   DATA[1858,0] := 2.531467;
   DATA[1858,1] := 861.0878;
   DATA[1858,2] := 2.0;
   DATA[1858,3] := 2.0;
   DATA[1858,4] := 263.362;
   DATA[1858,5] := 8.398359;
   DATA[1858,6] := 333.3761;
   DATA[1858,7] := 2.469228;
   DATA[1858,8] := 2.0;
   DATA[1858,9] := 2.0;
   DATA[1858,10] := 2.0;
   DATA[1858,11] := 19.80601;
   DATA[1858,12] := 2.208756;
   DATA[1858,13] := 790.5024;
   DATA[1858,14] := 1.0;
   DATA[1858,15] := 2.0;
   DATA[1858,16] := 1.0;
   DATA[1858,17] := 1.0;
   DATA[1858,18] := 1.0;
   DATA[1858,19] := 2.0;
   DATA[1858,20] := 148.808;
   DATA[1858,21] := 154.4476;
   DATA[1858,22] := 1.711723;
   DATA[1858,23] := 818.2517;
   DATA[1858,24] := 2.0;
   DATA[1858,25] := 2.0;
   DATA[1858,26] := 7.874135;
   DATA[1858,27] := 143.5529;
   DATA[1858,28] := 262.3686;
   DATA[1858,29] := 12.15073;
   DATA[1858,30] := 1.72161;
   DATA[1858,31] := 1.282567;
   DATA[1858,32] := 0.7355248;
   DATA[1858,33] := 0.3084265;
   DATA[1858,34] := 2.0;
   DATA[1858,35] := 249.8238;
   DATA[1858,36] := 1.69801;
   DATA[1858,37] := 188.6856;
   DATA[1858,38] := 0.000128152;
   DATA[1858,39] := 1.0;
   DATA[1858,40] := 1.0;
   DATA[1859,0] := 2.567658;
   DATA[1859,1] := 861.0093;
   DATA[1859,2] := 2.0;
   DATA[1859,3] := 2.0;
   DATA[1859,4] := 263.362;
   DATA[1859,5] := 8.398039;
   DATA[1859,6] := 333.4786;
   DATA[1859,7] := 2.469228;
   DATA[1859,8] := 2.0;
   DATA[1859,9] := 2.0;
   DATA[1859,10] := 2.0;
   DATA[1859,11] := 19.80601;
   DATA[1859,12] := 2.208756;
   DATA[1859,13] := 790.7027;
   DATA[1859,14] := 1.0;
   DATA[1859,15] := 2.0;
   DATA[1859,16] := 1.0;
   DATA[1859,17] := 1.0;
   DATA[1859,18] := 1.0;
   DATA[1859,19] := 2.0;
   DATA[1859,20] := 148.808;
   DATA[1859,21] := 154.4476;
   DATA[1859,22] := 1.710313;
   DATA[1859,23] := 818.2902;
   DATA[1859,24] := 2.0;
   DATA[1859,25] := 2.0;
   DATA[1859,26] := 7.874135;
   DATA[1859,27] := 143.5529;
   DATA[1859,28] := 262.3686;
   DATA[1859,29] := 12.15073;
   DATA[1859,30] := 1.72161;
   DATA[1859,31] := 1.273473;
   DATA[1859,32] := 0.7355248;
   DATA[1859,33] := 0.3084265;
   DATA[1859,34] := 2.0;
   DATA[1859,35] := 249.8238;
   DATA[1859,36] := 1.69801;
   DATA[1859,37] := 188.6856;
   DATA[1859,38] := 0.000128152;
   DATA[1859,39] := 1.0;
   DATA[1859,40] := 1.0;
   DATA[1860,0] := 2.606091;
   DATA[1860,1] := 860.6167;
   DATA[1860,2] := 2.0;
   DATA[1860,3] := 2.0;
   DATA[1860,4] := 263.2979;
   DATA[1860,5] := 8.393873;
   DATA[1860,6] := 333.4786;
   DATA[1860,7] := 2.469228;
   DATA[1860,8] := 2.0;
   DATA[1860,9] := 2.0;
   DATA[1860,10] := 2.0;
   DATA[1860,11] := 19.80601;
   DATA[1860,12] := 2.210294;
   DATA[1860,13] := 790.7027;
   DATA[1860,14] := 1.0;
   DATA[1860,15] := 2.0;
   DATA[1860,16] := 1.0;
   DATA[1860,17] := 1.0;
   DATA[1860,18] := 1.0;
   DATA[1860,19] := 2.0;
   DATA[1860,20] := 148.808;
   DATA[1860,21] := 154.4476;
   DATA[1860,22] := 1.710313;
   DATA[1860,23] := 818.2517;
   DATA[1860,24] := 2.0;
   DATA[1860,25] := 2.0;
   DATA[1860,26] := 7.874135;
   DATA[1860,27] := 143.5529;
   DATA[1860,28] := 262.3686;
   DATA[1860,29] := 12.15073;
   DATA[1860,30] := 1.723532;
   DATA[1860,31] := 1.277187;
   DATA[1860,32] := 0.7355248;
   DATA[1860,33] := 0.3084265;
   DATA[1860,34] := 2.0;
   DATA[1860,35] := 250.0961;
   DATA[1860,36] := 1.69801;
   DATA[1860,37] := 189.006;
   DATA[1860,38] := 0.000128152;
   DATA[1860,39] := 1.0;
   DATA[1860,40] := 1.0;
   DATA[1861,0] := 2.633635;
   DATA[1861,1] := 860.8522;
   DATA[1861,2] := 2.0;
   DATA[1861,3] := 2.0;
   DATA[1861,4] := 263.0095;
   DATA[1861,5] := 8.393873;
   DATA[1861,6] := 333.4786;
   DATA[1861,7] := 2.469228;
   DATA[1861,8] := 2.0;
   DATA[1861,9] := 2.0;
   DATA[1861,10] := 2.0;
   DATA[1861,11] := 19.73238;
   DATA[1861,12] := 2.210294;
   DATA[1861,13] := 790.7828;
   DATA[1861,14] := 1.0;
   DATA[1861,15] := 2.0;
   DATA[1861,16] := 1.0;
   DATA[1861,17] := 1.0;
   DATA[1861,18] := 1.0;
   DATA[1861,19] := 2.0;
   DATA[1861,20] := 148.808;
   DATA[1861,21] := 154.5245;
   DATA[1861,22] := 1.710313;
   DATA[1861,23] := 817.9441;
   DATA[1861,24] := 2.0;
   DATA[1861,25] := 2.0;
   DATA[1861,26] := 7.874135;
   DATA[1861,27] := 143.5529;
   DATA[1861,28] := 262.3686;
   DATA[1861,29] := 12.15073;
   DATA[1861,30] := 1.724045;
   DATA[1861,31] := 1.275522;
   DATA[1861,32] := 0.7355248;
   DATA[1861,33] := 0.3084265;
   DATA[1861,34] := 2.0;
   DATA[1861,35] := 250.0961;
   DATA[1861,36] := 1.69801;
   DATA[1861,37] := 189.006;
   DATA[1861,38] := 0.000128152;
   DATA[1861,39] := 1.0;
   DATA[1861,40] := 1.0;
   DATA[1862,0] := 2.654133;
   DATA[1862,1] := 860.8915;
   DATA[1862,2] := 2.0;
   DATA[1862,3] := 2.0;
   DATA[1862,4] := 262.9454;
   DATA[1862,5] := 8.393873;
   DATA[1862,6] := 333.4786;
   DATA[1862,7] := 2.469228;
   DATA[1862,8] := 2.0;
   DATA[1862,9] := 2.0;
   DATA[1862,10] := 2.0;
   DATA[1862,11] := 19.73238;
   DATA[1862,12] := 2.207731;
   DATA[1862,13] := 791.4637;
   DATA[1862,14] := 1.0;
   DATA[1862,15] := 2.0;
   DATA[1862,16] := 1.0;
   DATA[1862,17] := 1.0;
   DATA[1862,18] := 1.0;
   DATA[1862,19] := 2.0;
   DATA[1862,20] := 148.808;
   DATA[1862,21] := 154.5245;
   DATA[1862,22] := 1.710313;
   DATA[1862,23] := 818.4055;
   DATA[1862,24] := 2.0;
   DATA[1862,25] := 2.0;
   DATA[1862,26] := 7.874135;
   DATA[1862,27] := 143.5529;
   DATA[1862,28] := 262.3686;
   DATA[1862,29] := 12.15073;
   DATA[1862,30] := 1.724045;
   DATA[1862,31] := 1.278596;
   DATA[1862,32] := 0.7355248;
   DATA[1862,33] := 0.3084265;
   DATA[1862,34] := 2.0;
   DATA[1862,35] := 250.0961;
   DATA[1862,36] := 1.69801;
   DATA[1862,37] := 189.006;
   DATA[1862,38] := 0.000128152;
   DATA[1862,39] := 1.0;
   DATA[1862,40] := 1.0;
   DATA[1863,0] := 2.664382;
   DATA[1863,1] := 860.8915;
   DATA[1863,2] := 2.0;
   DATA[1863,3] := 2.0;
   DATA[1863,4] := 262.9454;
   DATA[1863,5] := 8.393873;
   DATA[1863,6] := 333.4786;
   DATA[1863,7] := 2.469228;
   DATA[1863,8] := 2.0;
   DATA[1863,9] := 2.0;
   DATA[1863,10] := 2.0;
   DATA[1863,11] := 19.73238;
   DATA[1863,12] := 2.20581;
   DATA[1863,13] := 791.664;
   DATA[1863,14] := 1.0;
   DATA[1863,15] := 2.0;
   DATA[1863,16] := 1.0;
   DATA[1863,17] := 1.0;
   DATA[1863,18] := 1.0;
   DATA[1863,19] := 2.0;
   DATA[1863,20] := 148.808;
   DATA[1863,21] := 154.5245;
   DATA[1863,22] := 1.710313;
   DATA[1863,23] := 818.444;
   DATA[1863,24] := 2.0;
   DATA[1863,25] := 2.0;
   DATA[1863,26] := 7.874135;
   DATA[1863,27] := 143.5529;
   DATA[1863,28] := 262.3686;
   DATA[1863,29] := 12.15073;
   DATA[1863,30] := 1.724045;
   DATA[1863,31] := 1.291405;
   DATA[1863,32] := 0.7355248;
   DATA[1863,33] := 0.3084265;
   DATA[1863,34] := 2.0;
   DATA[1863,35] := 250.0961;
   DATA[1863,36] := 1.69801;
   DATA[1863,37] := 189.006;
   DATA[1863,38] := 0.000128152;
   DATA[1863,39] := 1.0;
   DATA[1863,40] := 1.0;
   DATA[1864,0] := 2.664382;
   DATA[1864,1] := 861.127;
   DATA[1864,2] := 2.0;
   DATA[1864,3] := 2.0;
   DATA[1864,4] := 262.9454;
   DATA[1864,5] := 8.393873;
   DATA[1864,6] := 333.4786;
   DATA[1864,7] := 2.467818;
   DATA[1864,8] := 2.0;
   DATA[1864,9] := 2.0;
   DATA[1864,10] := 2.0;
   DATA[1864,11] := 19.73238;
   DATA[1864,12] := 2.20581;
   DATA[1864,13] := 791.9044;
   DATA[1864,14] := 1.0;
   DATA[1864,15] := 2.0;
   DATA[1864,16] := 1.0;
   DATA[1864,17] := 1.0;
   DATA[1864,18] := 1.0;
   DATA[1864,19] := 2.0;
   DATA[1864,20] := 148.808;
   DATA[1864,21] := 154.5245;
   DATA[1864,22] := 1.710313;
   DATA[1864,23] := 818.6747;
   DATA[1864,24] := 2.0;
   DATA[1864,25] := 2.0;
   DATA[1864,26] := 7.874135;
   DATA[1864,27] := 143.5529;
   DATA[1864,28] := 262.3045;
   DATA[1864,29] := 12.15073;
   DATA[1864,30] := 1.724045;
   DATA[1864,31] := 1.28641;
   DATA[1864,32] := 0.7355248;
   DATA[1864,33] := 0.3084265;
   DATA[1864,34] := 2.0;
   DATA[1864,35] := 250.0961;
   DATA[1864,36] := 1.537821;
   DATA[1864,37] := 188.8618;
   DATA[1864,38] := 0.000128152;
   DATA[1864,39] := 1.0;
   DATA[1864,40] := 1.0;
   DATA[1865,0] := 2.63876;
   DATA[1865,1] := 861.2055;
   DATA[1865,2] := 2.0;
   DATA[1865,3] := 2.0;
   DATA[1865,4] := 262.9454;
   DATA[1865,5] := 8.393873;
   DATA[1865,6] := 333.6837;
   DATA[1865,7] := 2.467818;
   DATA[1865,8] := 2.0;
   DATA[1865,9] := 2.0;
   DATA[1865,10] := 2.0;
   DATA[1865,11] := 19.73238;
   DATA[1865,12] := 2.208244;
   DATA[1865,13] := 791.9044;
   DATA[1865,14] := 1.0;
   DATA[1865,15] := 2.0;
   DATA[1865,16] := 1.0;
   DATA[1865,17] := 1.0;
   DATA[1865,18] := 1.0;
   DATA[1865,19] := 2.0;
   DATA[1865,20] := 148.808;
   DATA[1865,21] := 154.5245;
   DATA[1865,22] := 1.710698;
   DATA[1865,23] := 819.213;
   DATA[1865,24] := 2.0;
   DATA[1865,25] := 2.0;
   DATA[1865,26] := 7.874135;
   DATA[1865,27] := 143.5529;
   DATA[1865,28] := 262.1764;
   DATA[1865,29] := 12.15073;
   DATA[1865,30] := 1.724045;
   DATA[1865,31] := 1.289356;
   DATA[1865,32] := 0.7355248;
   DATA[1865,33] := 0.3084265;
   DATA[1865,34] := 2.0;
   DATA[1865,35] := 250.0961;
   DATA[1865,36] := 1.537821;
   DATA[1865,37] := 188.6856;
   DATA[1865,38] := 0.000128152;
   DATA[1865,39] := 1.0;
   DATA[1865,40] := 1.0;
   DATA[1866,0] := 2.630753;
   DATA[1866,1] := 860.8915;
   DATA[1866,2] := 2.0;
   DATA[1866,3] := 2.0;
   DATA[1866,4] := 262.9454;
   DATA[1866,5] := 8.393873;
   DATA[1866,6] := 333.6837;
   DATA[1866,7] := 2.467818;
   DATA[1866,8] := 2.0;
   DATA[1866,9] := 2.0;
   DATA[1866,10] := 2.0;
   DATA[1866,11] := 19.73238;
   DATA[1866,12] := 2.209397;
   DATA[1866,13] := 792.0646;
   DATA[1866,14] := 1.0;
   DATA[1866,15] := 2.0;
   DATA[1866,16] := 1.0;
   DATA[1866,17] := 1.0;
   DATA[1866,18] := 1.0;
   DATA[1866,19] := 2.0;
   DATA[1866,20] := 148.808;
   DATA[1866,21] := 154.6526;
   DATA[1866,22] := 1.712107;
   DATA[1866,23] := 818.9823;
   DATA[1866,24] := 2.0;
   DATA[1866,25] := 2.0;
   DATA[1866,26] := 7.874135;
   DATA[1866,27] := 143.5529;
   DATA[1866,28] := 262.1764;
   DATA[1866,29] := 12.15073;
   DATA[1866,30] := 1.724045;
   DATA[1866,31] := 1.291789;
   DATA[1866,32] := 0.7355248;
   DATA[1866,33] := 0.3084265;
   DATA[1866,34] := 2.0;
   DATA[1866,35] := 250.0961;
   DATA[1866,36] := 1.762086;
   DATA[1866,37] := 188.6856;
   DATA[1866,38] := 0.000128152;
   DATA[1866,39] := 1.0;
   DATA[1866,40] := 1.0;
   DATA[1867,0] := 2.625628;
   DATA[1867,1] := 861.0878;
   DATA[1867,2] := 2.0;
   DATA[1867,3] := 2.0;
   DATA[1867,4] := 262.9454;
   DATA[1867,5] := 8.393873;
   DATA[1867,6] := 333.6837;
   DATA[1867,7] := 2.467818;
   DATA[1867,8] := 2.0;
   DATA[1867,9] := 2.0;
   DATA[1867,10] := 2.0;
   DATA[1867,11] := 19.69396;
   DATA[1867,12] := 2.209397;
   DATA[1867,13] := 792.3449;
   DATA[1867,14] := 1.0;
   DATA[1867,15] := 2.0;
   DATA[1867,16] := 1.0;
   DATA[1867,17] := 1.0;
   DATA[1867,18] := 1.0;
   DATA[1867,19] := 2.0;
   DATA[1867,20] := 148.808;
   DATA[1867,21] := 154.6526;
   DATA[1867,22] := 1.714286;
   DATA[1867,23] := 819.1746;
   DATA[1867,24] := 2.0;
   DATA[1867,25] := 2.0;
   DATA[1867,26] := 7.874135;
   DATA[1867,27] := 143.5529;
   DATA[1867,28] := 262.1764;
   DATA[1867,29] := 12.15073;
   DATA[1867,30] := 1.723789;
   DATA[1867,31] := 1.293455;
   DATA[1867,32] := 0.7355248;
   DATA[1867,33] := 0.3084265;
   DATA[1867,34] := 2.0;
   DATA[1867,35] := 250.0961;
   DATA[1867,36] := 1.762086;
   DATA[1867,37] := 188.6856;
   DATA[1867,38] := 0.000128152;
   DATA[1867,39] := 1.0;
   DATA[1867,40] := 1.0;
   DATA[1868,0] := 2.617942;
   DATA[1868,1] := 860.813;
   DATA[1868,2] := 2.0;
   DATA[1868,3] := 2.0;
   DATA[1868,4] := 262.9454;
   DATA[1868,5] := 8.393873;
   DATA[1868,6] := 333.6837;
   DATA[1868,7] := 2.467818;
   DATA[1868,8] := 2.0;
   DATA[1868,9] := 2.0;
   DATA[1868,10] := 2.0;
   DATA[1868,11] := 19.69396;
   DATA[1868,12] := 2.209397;
   DATA[1868,13] := 792.3049;
   DATA[1868,14] := 1.0;
   DATA[1868,15] := 2.0;
   DATA[1868,16] := 1.0;
   DATA[1868,17] := 1.0;
   DATA[1868,18] := 1.0;
   DATA[1868,19] := 2.0;
   DATA[1868,20] := 148.808;
   DATA[1868,21] := 154.6526;
   DATA[1868,22] := 1.714926;
   DATA[1868,23] := 819.0977;
   DATA[1868,24] := 2.0;
   DATA[1868,25] := 2.0;
   DATA[1868,26] := 7.874135;
   DATA[1868,27] := 143.5529;
   DATA[1868,28] := 262.1764;
   DATA[1868,29] := 12.15073;
   DATA[1868,30] := 1.721866;
   DATA[1868,31] := 1.302165;
   DATA[1868,32] := 0.7355248;
   DATA[1868,33] := 0.3084265;
   DATA[1868,34] := 2.0;
   DATA[1868,35] := 249.9359;
   DATA[1868,36] := 1.762086;
   DATA[1868,37] := 188.8618;
   DATA[1868,38] := 0.000128152;
   DATA[1868,39] := 1.0;
   DATA[1868,40] := 1.0;
   DATA[1869,0] := 2.596483;
   DATA[1869,1] := 860.6167;
   DATA[1869,2] := 2.0;
   DATA[1869,3] := 2.0;
   DATA[1869,4] := 262.9454;
   DATA[1869,5] := 8.393873;
   DATA[1869,6] := 333.6837;
   DATA[1869,7] := 2.467818;
   DATA[1869,8] := 2.0;
   DATA[1869,9] := 2.0;
   DATA[1869,10] := 2.0;
   DATA[1869,11] := 19.71637;
   DATA[1869,12] := 2.209397;
   DATA[1869,13] := 792.6653;
   DATA[1869,14] := 1.0;
   DATA[1869,15] := 2.0;
   DATA[1869,16] := 1.0;
   DATA[1869,17] := 1.0;
   DATA[1869,18] := 1.0;
   DATA[1869,19] := 2.0;
   DATA[1869,20] := 148.808;
   DATA[1869,21] := 154.6526;
   DATA[1869,22] := 1.714926;
   DATA[1869,23] := 819.6744;
   DATA[1869,24] := 2.0;
   DATA[1869,25] := 2.0;
   DATA[1869,26] := 7.874135;
   DATA[1869,27] := 143.5529;
   DATA[1869,28] := 262.3366;
   DATA[1869,29] := 12.15073;
   DATA[1869,30] := 1.721866;
   DATA[1869,31] := 1.29512;
   DATA[1869,32] := 0.7355248;
   DATA[1869,33] := 0.3084265;
   DATA[1869,34] := 2.0;
   DATA[1869,35] := 249.9359;
   DATA[1869,36] := 1.762086;
   DATA[1869,37] := 188.8618;
   DATA[1869,38] := 0.000128152;
   DATA[1869,39] := 1.0;
   DATA[1869,40] := 1.0;
   DATA[1870,0] := 2.58111;
   DATA[1870,1] := 860.4205;
   DATA[1870,2] := 2.0;
   DATA[1870,3] := 2.0;
   DATA[1870,4] := 262.9454;
   DATA[1870,5] := 8.392271;
   DATA[1870,6] := 333.4786;
   DATA[1870,7] := 2.46769;
   DATA[1870,8] := 2.0;
   DATA[1870,9] := 2.0;
   DATA[1870,10] := 2.0;
   DATA[1870,11] := 19.73878;
   DATA[1870,12] := 2.209397;
   DATA[1870,13] := 793.146;
   DATA[1870,14] := 1.0;
   DATA[1870,15] := 2.0;
   DATA[1870,16] := 1.0;
   DATA[1870,17] := 1.0;
   DATA[1870,18] := 1.0;
   DATA[1870,19] := 2.0;
   DATA[1870,20] := 148.808;
   DATA[1870,21] := 154.6526;
   DATA[1870,22] := 1.714926;
   DATA[1870,23] := 819.5591;
   DATA[1870,24] := 2.0;
   DATA[1870,25] := 2.0;
   DATA[1870,26] := 7.874135;
   DATA[1870,27] := 143.5529;
   DATA[1870,28] := 262.3366;
   DATA[1870,29] := 12.15073;
   DATA[1870,30] := 1.724045;
   DATA[1870,31] := 1.292174;
   DATA[1870,32] := 0.7355248;
   DATA[1870,33] := 0.3084265;
   DATA[1870,34] := 2.0;
   DATA[1870,35] := 249.9359;
   DATA[1870,36] := 1.762086;
   DATA[1870,37] := 188.8618;
   DATA[1870,38] := 0.000128152;
   DATA[1870,39] := 1.0;
   DATA[1870,40] := 1.0;
   DATA[1871,0] := 2.55837;
   DATA[1871,1] := 860.2634;
   DATA[1871,2] := 2.0;
   DATA[1871,3] := 2.0;
   DATA[1871,4] := 262.9454;
   DATA[1871,5] := 8.39163;
   DATA[1871,6] := 333.4273;
   DATA[1871,7] := 2.466024;
   DATA[1871,8] := 2.0;
   DATA[1871,9] := 2.0;
   DATA[1871,10] := 2.0;
   DATA[1871,11] := 19.73878;
   DATA[1871,12] := 2.21119;
   DATA[1871,13] := 793.0659;
   DATA[1871,14] := 1.0;
   DATA[1871,15] := 2.0;
   DATA[1871,16] := 1.0;
   DATA[1871,17] := 1.0;
   DATA[1871,18] := 1.0;
   DATA[1871,19] := 2.0;
   DATA[1871,20] := 148.808;
   DATA[1871,21] := 154.6526;
   DATA[1871,22] := 1.717105;
   DATA[1871,23] := 819.213;
   DATA[1871,24] := 2.0;
   DATA[1871,25] := 2.0;
   DATA[1871,26] := 7.874135;
   DATA[1871,27] := 143.5529;
   DATA[1871,28] := 262.3366;
   DATA[1871,29] := 12.15073;
   DATA[1871,30] := 1.724173;
   DATA[1871,31] := 1.290637;
   DATA[1871,32] := 0.7355248;
   DATA[1871,33] := 0.3084265;
   DATA[1871,34] := 2.0;
   DATA[1871,35] := 249.9359;
   DATA[1871,36] := 1.762086;
   DATA[1871,37] := 188.8618;
   DATA[1871,38] := 0.000128152;
   DATA[1871,39] := 1.0;
   DATA[1871,40] := 1.0;
   DATA[1872,0] := 2.542356;
   DATA[1872,1] := 860.4205;
   DATA[1872,2] := 2.0;
   DATA[1872,3] := 2.0;
   DATA[1872,4] := 262.9454;
   DATA[1872,5] := 8.39163;
   DATA[1872,6] := 333.4273;
   DATA[1872,7] := 2.466024;
   DATA[1872,8] := 2.0;
   DATA[1872,9] := 2.0;
   DATA[1872,10] := 2.0;
   DATA[1872,11] := 19.73878;
   DATA[1872,12] := 2.21119;
   DATA[1872,13] := 793.3062;
   DATA[1872,14] := 1.0;
   DATA[1872,15] := 2.0;
   DATA[1872,16] := 1.0;
   DATA[1872,17] := 1.0;
   DATA[1872,18] := 1.0;
   DATA[1872,19] := 2.0;
   DATA[1872,20] := 148.808;
   DATA[1872,21] := 154.6526;
   DATA[1872,22] := 1.717105;
   DATA[1872,23] := 819.4053;
   DATA[1872,24] := 2.0;
   DATA[1872,25] := 2.0;
   DATA[1872,26] := 7.874135;
   DATA[1872,27] := 143.5529;
   DATA[1872,28] := 262.3366;
   DATA[1872,29] := 12.15073;
   DATA[1872,30] := 1.724173;
   DATA[1872,31] := 1.282183;
   DATA[1872,32] := 0.7355248;
   DATA[1872,33] := 0.3084265;
   DATA[1872,34] := 2.0;
   DATA[1872,35] := 250.1442;
   DATA[1872,36] := 1.762086;
   DATA[1872,37] := 189.0861;
   DATA[1872,38] := 0.000128152;
   DATA[1872,39] := 1.0;
   DATA[1872,40] := 1.0;
   DATA[1873,0] := 2.521538;
   DATA[1873,1] := 860.4205;
   DATA[1873,2] := 2.0;
   DATA[1873,3] := 2.0;
   DATA[1873,4] := 262.9454;
   DATA[1873,5] := 8.39163;
   DATA[1873,6] := 333.4273;
   DATA[1873,7] := 2.466024;
   DATA[1873,8] := 2.0;
   DATA[1873,9] := 2.0;
   DATA[1873,10] := 2.0;
   DATA[1873,11] := 19.73878;
   DATA[1873,12] := 2.209909;
   DATA[1873,13] := 793.146;
   DATA[1873,14] := 1.0;
   DATA[1873,15] := 2.0;
   DATA[1873,16] := 1.0;
   DATA[1873,17] := 1.0;
   DATA[1873,18] := 1.0;
   DATA[1873,19] := 2.0;
   DATA[1873,20] := 148.808;
   DATA[1873,21] := 154.6526;
   DATA[1873,22] := 1.717105;
   DATA[1873,23] := 819.5975;
   DATA[1873,24] := 2.0;
   DATA[1873,25] := 2.0;
   DATA[1873,26] := 7.874135;
   DATA[1873,27] := 143.5529;
   DATA[1873,28] := 262.3366;
   DATA[1873,29] := 12.03538;
   DATA[1873,30] := 1.724686;
   DATA[1873,31] := 1.291277;
   DATA[1873,32] := 0.7355248;
   DATA[1873,33] := 0.3084265;
   DATA[1873,34] := 2.0;
   DATA[1873,35] := 250.1442;
   DATA[1873,36] := 1.762086;
   DATA[1873,37] := 189.0861;
   DATA[1873,38] := 0.000128152;
   DATA[1873,39] := 1.0;
   DATA[1873,40] := 1.0;
   DATA[1874,0] := 2.504884;
   DATA[1874,1] := 860.5382;
   DATA[1874,2] := 2.0;
   DATA[1874,3] := 2.0;
   DATA[1874,4] := 262.9454;
   DATA[1874,5] := 8.39163;
   DATA[1874,6] := 333.4273;
   DATA[1874,7] := 2.466024;
   DATA[1874,8] := 2.0;
   DATA[1874,9] := 2.0;
   DATA[1874,10] := 2.0;
   DATA[1874,11] := 19.73878;
   DATA[1874,12] := 2.209909;
   DATA[1874,13] := 792.9858;
   DATA[1874,14] := 1.0;
   DATA[1874,15] := 2.0;
   DATA[1874,16] := 1.0;
   DATA[1874,17] := 1.0;
   DATA[1874,18] := 1.0;
   DATA[1874,19] := 2.0;
   DATA[1874,20] := 148.808;
   DATA[1874,21] := 154.6526;
   DATA[1874,22] := 1.717105;
   DATA[1874,23] := 819.5975;
   DATA[1874,24] := 2.0;
   DATA[1874,25] := 2.0;
   DATA[1874,26] := 7.874135;
   DATA[1874,27] := 143.5529;
   DATA[1874,28] := 262.3366;
   DATA[1874,29] := 12.03538;
   DATA[1874,30] := 1.725327;
   DATA[1874,31] := 1.29243;
   DATA[1874,32] := 0.7355248;
   DATA[1874,33] := 0.3084265;
   DATA[1874,34] := 2.0;
   DATA[1874,35] := 250.1442;
   DATA[1874,36] := 1.762086;
   DATA[1874,37] := 189.0861;
   DATA[1874,38] := 0.000128152;
   DATA[1874,39] := 1.0;
   DATA[1874,40] := 1.0;
   DATA[1875,0] := 2.489511;
   DATA[1875,1] := 860.7345;
   DATA[1875,2] := 2.0;
   DATA[1875,3] := 2.0;
   DATA[1875,4] := 262.8813;
   DATA[1875,5] := 8.39163;
   DATA[1875,6] := 333.4273;
   DATA[1875,7] := 2.466024;
   DATA[1875,8] := 2.0;
   DATA[1875,9] := 2.0;
   DATA[1875,10] := 2.0;
   DATA[1875,11] := 19.73878;
   DATA[1875,12] := 2.209653;
   DATA[1875,13] := 793.0659;
   DATA[1875,14] := 1.0;
   DATA[1875,15] := 2.0;
   DATA[1875,16] := 1.0;
   DATA[1875,17] := 1.0;
   DATA[1875,18] := 1.0;
   DATA[1875,19] := 2.0;
   DATA[1875,20] := 148.808;
   DATA[1875,21] := 154.6526;
   DATA[1875,22] := 1.716464;
   DATA[1875,23] := 819.5591;
   DATA[1875,24] := 2.0;
   DATA[1875,25] := 2.0;
   DATA[1875,26] := 7.874135;
   DATA[1875,27] := 143.5529;
   DATA[1875,28] := 262.3366;
   DATA[1875,29] := 12.03538;
   DATA[1875,30] := 1.725583;
   DATA[1875,31] := 1.295888;
   DATA[1875,32] := 0.7355248;
   DATA[1875,33] := 0.3084265;
   DATA[1875,34] := 2.0;
   DATA[1875,35] := 250.1442;
   DATA[1875,36] := 1.762086;
   DATA[1875,37] := 189.0861;
   DATA[1875,38] := 0.000128152;
   DATA[1875,39] := 1.0;
   DATA[1875,40] := 1.0;
   DATA[1876,0] := 2.484707;
   DATA[1876,1] := 860.3027;
   DATA[1876,2] := 2.0;
   DATA[1876,3] := 2.0;
   DATA[1876,4] := 262.8813;
   DATA[1876,5] := 8.39163;
   DATA[1876,6] := 333.4017;
   DATA[1876,7] := 2.466793;
   DATA[1876,8] := 2.0;
   DATA[1876,9] := 2.0;
   DATA[1876,10] := 2.0;
   DATA[1876,11] := 19.73878;
   DATA[1876,12] := 2.208756;
   DATA[1876,13] := 792.5853;
   DATA[1876,14] := 1.0;
   DATA[1876,15] := 2.0;
   DATA[1876,16] := 1.0;
   DATA[1876,17] := 1.0;
   DATA[1876,18] := 1.0;
   DATA[1876,19] := 2.0;
   DATA[1876,20] := 148.808;
   DATA[1876,21] := 154.6526;
   DATA[1876,22] := 1.714158;
   DATA[1876,23] := 819.6744;
   DATA[1876,24] := 2.0;
   DATA[1876,25] := 2.0;
   DATA[1876,26] := 7.874135;
   DATA[1876,27] := 143.6811;
   DATA[1876,28] := 262.3366;
   DATA[1876,29] := 12.03538;
   DATA[1876,30] := 1.726993;
   DATA[1876,31] := 1.302293;
   DATA[1876,32] := 0.7355248;
   DATA[1876,33] := 0.3084265;
   DATA[1876,34] := 2.0;
   DATA[1876,35] := 250.1442;
   DATA[1876,36] := 1.762086;
   DATA[1876,37] := 189.0861;
   DATA[1876,38] := 0.000128152;
   DATA[1876,39] := 1.0;
   DATA[1876,40] := 1.0;
   DATA[1877,0] := 2.46581;
   DATA[1877,1] := 860.2242;
   DATA[1877,2] := 2.0;
   DATA[1877,3] := 2.0;
   DATA[1877,4] := 262.8813;
   DATA[1877,5] := 8.39163;
   DATA[1877,6] := 333.3504;
   DATA[1877,7] := 2.466793;
   DATA[1877,8] := 2.0;
   DATA[1877,9] := 2.0;
   DATA[1877,10] := 2.0;
   DATA[1877,11] := 19.70037;
   DATA[1877,12] := 2.208756;
   DATA[1877,13] := 792.3449;
   DATA[1877,14] := 1.0;
   DATA[1877,15] := 2.0;
   DATA[1877,16] := 1.0;
   DATA[1877,17] := 1.0;
   DATA[1877,18] := 1.0;
   DATA[1877,19] := 2.0;
   DATA[1877,20] := 148.808;
   DATA[1877,21] := 154.6526;
   DATA[1877,22] := 1.714029;
   DATA[1877,23] := 819.5591;
   DATA[1877,24] := 2.0;
   DATA[1877,25] := 2.0;
   DATA[1877,26] := 7.874135;
   DATA[1877,27] := 143.6811;
   DATA[1877,28] := 262.3366;
   DATA[1877,29] := 12.03538;
   DATA[1877,30] := 1.727506;
   DATA[1877,31] := 1.302805;
   DATA[1877,32] := 0.7355248;
   DATA[1877,33] := 0.3084265;
   DATA[1877,34] := 2.0;
   DATA[1877,35] := 250.1442;
   DATA[1877,36] := 1.762086;
   DATA[1877,37] := 188.9419;
   DATA[1877,38] := 0.000128152;
   DATA[1877,39] := 1.0;
   DATA[1877,40] := 1.0;
   DATA[1878,0] := 2.457163;
   DATA[1878,1] := 859.9102;
   DATA[1878,2] := 2.0;
   DATA[1878,3] := 2.0;
   DATA[1878,4] := 262.8813;
   DATA[1878,5] := 8.39163;
   DATA[1878,6] := 333.2479;
   DATA[1878,7] := 2.466793;
   DATA[1878,8] := 2.0;
   DATA[1878,9] := 2.0;
   DATA[1878,10] := 2.0;
   DATA[1878,11] := 19.70037;
   DATA[1878,12] := 2.208756;
   DATA[1878,13] := 792.0646;
   DATA[1878,14] := 1.0;
   DATA[1878,15] := 2.0;
   DATA[1878,16] := 1.0;
   DATA[1878,17] := 1.0;
   DATA[1878,18] := 1.0;
   DATA[1878,19] := 2.0;
   DATA[1878,20] := 148.808;
   DATA[1878,21] := 154.6526;
   DATA[1878,22] := 1.714029;
   DATA[1878,23] := 819.7513;
   DATA[1878,24] := 2.0;
   DATA[1878,25] := 2.0;
   DATA[1878,26] := 7.874135;
   DATA[1878,27] := 143.6811;
   DATA[1878,28] := 262.3366;
   DATA[1878,29] := 12.03538;
   DATA[1878,30] := 1.727506;
   DATA[1878,31] := 1.302805;
   DATA[1878,32] := 0.7355248;
   DATA[1878,33] := 0.3084265;
   DATA[1878,34] := 2.0;
   DATA[1878,35] := 250.1442;
   DATA[1878,36] := 1.762086;
   DATA[1878,37] := 188.8939;
   DATA[1878,38] := 0.000128152;
   DATA[1878,39] := 1.0;
   DATA[1878,40] := 1.0;
   DATA[1879,0] := 2.441469;
   DATA[1879,1] := 859.8709;
   DATA[1879,2] := 2.0;
   DATA[1879,3] := 2.0;
   DATA[1879,4] := 262.8813;
   DATA[1879,5] := 8.39163;
   DATA[1879,6] := 333.2479;
   DATA[1879,7] := 2.466793;
   DATA[1879,8] := 2.0;
   DATA[1879,9] := 2.0;
   DATA[1879,10] := 2.0;
   DATA[1879,11] := 19.70037;
   DATA[1879,12] := 2.208756;
   DATA[1879,13] := 792.1847;
   DATA[1879,14] := 1.0;
   DATA[1879,15] := 2.0;
   DATA[1879,16] := 1.0;
   DATA[1879,17] := 1.0;
   DATA[1879,18] := 1.0;
   DATA[1879,19] := 2.0;
   DATA[1879,20] := 148.808;
   DATA[1879,21] := 154.6526;
   DATA[1879,22] := 1.714029;
   DATA[1879,23] := 819.6744;
   DATA[1879,24] := 2.0;
   DATA[1879,25] := 2.0;
   DATA[1879,26] := 7.874135;
   DATA[1879,27] := 143.6811;
   DATA[1879,28] := 262.3366;
   DATA[1879,29] := 12.03538;
   DATA[1879,30] := 1.727506;
   DATA[1879,31] := 1.300243;
   DATA[1879,32] := 0.7355248;
   DATA[1879,33] := 0.3084265;
   DATA[1879,34] := 2.0;
   DATA[1879,35] := 250.1442;
   DATA[1879,36] := 1.762086;
   DATA[1879,37] := 188.8939;
   DATA[1879,38] := 0.000128152;
   DATA[1879,39] := 1.0;
   DATA[1879,40] := 1.0;
   DATA[1880,0] := 2.428338;
   DATA[1880,1] := 859.4784;
   DATA[1880,2] := 2.0;
   DATA[1880,3] := 2.0;
   DATA[1880,4] := 262.8813;
   DATA[1880,5] := 8.39163;
   DATA[1880,6] := 333.2479;
   DATA[1880,7] := 2.466793;
   DATA[1880,8] := 2.0;
   DATA[1880,9] := 2.0;
   DATA[1880,10] := 2.0;
   DATA[1880,11] := 19.72598;
   DATA[1880,12] := 2.209269;
   DATA[1880,13] := 792.2648;
   DATA[1880,14] := 1.0;
   DATA[1880,15] := 2.0;
   DATA[1880,16] := 1.0;
   DATA[1880,17] := 1.0;
   DATA[1880,18] := 1.0;
   DATA[1880,19] := 2.0;
   DATA[1880,20] := 148.808;
   DATA[1880,21] := 154.6783;
   DATA[1880,22] := 1.714029;
   DATA[1880,23] := 819.636;
   DATA[1880,24] := 2.0;
   DATA[1880,25] := 2.0;
   DATA[1880,26] := 7.874135;
   DATA[1880,27] := 143.6811;
   DATA[1880,28] := 262.3366;
   DATA[1880,29] := 12.03538;
   DATA[1880,30] := 1.726865;
   DATA[1880,31] := 1.29243;
   DATA[1880,32] := 0.7355248;
   DATA[1880,33] := 0.3084265;
   DATA[1880,34] := 2.0;
   DATA[1880,35] := 250.1442;
   DATA[1880,36] := 1.762086;
   DATA[1880,37] := 188.8939;
   DATA[1880,38] := 0.000128152;
   DATA[1880,39] := 1.0;
   DATA[1880,40] := 1.0;
   DATA[1881,0] := 2.428338;
   DATA[1881,1] := 859.2821;
   DATA[1881,2] := 2.0;
   DATA[1881,3] := 2.0;
   DATA[1881,4] := 262.6891;
   DATA[1881,5] := 8.39163;
   DATA[1881,6] := 333.2479;
   DATA[1881,7] := 2.466793;
   DATA[1881,8] := 2.0;
   DATA[1881,9] := 2.0;
   DATA[1881,10] := 2.0;
   DATA[1881,11] := 19.72598;
   DATA[1881,12] := 2.209269;
   DATA[1881,13] := 792.1847;
   DATA[1881,14] := 1.0;
   DATA[1881,15] := 2.0;
   DATA[1881,16] := 1.0;
   DATA[1881,17] := 1.0;
   DATA[1881,18] := 1.0;
   DATA[1881,19] := 2.0;
   DATA[1881,20] := 148.808;
   DATA[1881,21] := 154.7552;
   DATA[1881,22] := 1.714029;
   DATA[1881,23] := 819.7898;
   DATA[1881,24] := 2.0;
   DATA[1881,25] := 2.0;
   DATA[1881,26] := 7.874135;
   DATA[1881,27] := 143.6811;
   DATA[1881,28] := 262.3366;
   DATA[1881,29] := 12.03538;
   DATA[1881,30] := 1.726224;
   DATA[1881,31] := 1.298834;
   DATA[1881,32] := 0.7355248;
   DATA[1881,33] := 0.3084265;
   DATA[1881,34] := 2.0;
   DATA[1881,35] := 250.1442;
   DATA[1881,36] := 1.649953;
   DATA[1881,37] := 188.8939;
   DATA[1881,38] := 0.000128152;
   DATA[1881,39] := 1.0;
   DATA[1881,40] := 1.0;
   DATA[1882,0] := 2.428338;
   DATA[1882,1] := 859.2429;
   DATA[1882,2] := 2.0;
   DATA[1882,3] := 2.0;
   DATA[1882,4] := 262.6891;
   DATA[1882,5] := 8.39163;
   DATA[1882,6] := 333.2479;
   DATA[1882,7] := 2.464486;
   DATA[1882,8] := 2.0;
   DATA[1882,9] := 2.0;
   DATA[1882,10] := 2.0;
   DATA[1882,11] := 19.72598;
   DATA[1882,12] := 2.209269;
   DATA[1882,13] := 792.1447;
   DATA[1882,14] := 1.0;
   DATA[1882,15] := 2.0;
   DATA[1882,16] := 1.0;
   DATA[1882,17] := 1.0;
   DATA[1882,18] := 1.0;
   DATA[1882,19] := 2.0;
   DATA[1882,20] := 148.808;
   DATA[1882,21] := 154.7552;
   DATA[1882,22] := 1.714029;
   DATA[1882,23] := 819.8282;
   DATA[1882,24] := 2.0;
   DATA[1882,25] := 2.0;
   DATA[1882,26] := 7.874135;
   DATA[1882,27] := 143.6811;
   DATA[1882,28] := 262.3366;
   DATA[1882,29] := 12.03538;
   DATA[1882,30] := 1.724942;
   DATA[1882,31] := 1.289996;
   DATA[1882,32] := 0.7355248;
   DATA[1882,33] := 0.3084265;
   DATA[1882,34] := 2.0;
   DATA[1882,35] := 250.1442;
   DATA[1882,36] := 1.649953;
   DATA[1882,37] := 188.8939;
   DATA[1882,38] := 0.000128152;
   DATA[1882,39] := 1.0;
   DATA[1882,40] := 1.0;
   DATA[1883,0] := 2.455562;
   DATA[1883,1] := 859.6747;
   DATA[1883,2] := 2.0;
   DATA[1883,3] := 2.0;
   DATA[1883,4] := 262.6891;
   DATA[1883,5] := 8.39163;
   DATA[1883,6] := 333.2479;
   DATA[1883,7] := 2.463589;
   DATA[1883,8] := 2.0;
   DATA[1883,9] := 2.0;
   DATA[1883,10] := 2.0;
   DATA[1883,11] := 19.72598;
   DATA[1883,12] := 2.209269;
   DATA[1883,13] := 792.3449;
   DATA[1883,14] := 1.0;
   DATA[1883,15] := 2.0;
   DATA[1883,16] := 1.0;
   DATA[1883,17] := 1.0;
   DATA[1883,18] := 1.0;
   DATA[1883,19] := 2.0;
   DATA[1883,20] := 148.808;
   DATA[1883,21] := 154.7552;
   DATA[1883,22] := 1.71608;
   DATA[1883,23] := 820.1743;
   DATA[1883,24] := 2.0;
   DATA[1883,25] := 2.0;
   DATA[1883,26] := 7.874135;
   DATA[1883,27] := 143.6811;
   DATA[1883,28] := 262.3366;
   DATA[1883,29] := 12.03538;
   DATA[1883,30] := 1.724942;
   DATA[1883,31] := 1.27296;
   DATA[1883,32] := 0.7355248;
   DATA[1883,33] := 0.3084265;
   DATA[1883,34] := 2.0;
   DATA[1883,35] := 250.032;
   DATA[1883,36] := 1.649953;
   DATA[1883,37] := 188.8939;
   DATA[1883,38] := 0.000128152;
   DATA[1883,39] := 1.0;
   DATA[1883,40] := 1.0;
   DATA[1884,0] := 2.500721;
   DATA[1884,1] := 859.0466;
   DATA[1884,2] := 2.0;
   DATA[1884,3] := 2.0;
   DATA[1884,4] := 262.6891;
   DATA[1884,5] := 8.39163;
   DATA[1884,6] := 333.2479;
   DATA[1884,7] := 2.463589;
   DATA[1884,8] := 2.0;
   DATA[1884,9] := 2.0;
   DATA[1884,10] := 2.0;
   DATA[1884,11] := 19.72598;
   DATA[1884,12] := 2.207603;
   DATA[1884,13] := 792.1447;
   DATA[1884,14] := 1.0;
   DATA[1884,15] := 2.0;
   DATA[1884,16] := 1.0;
   DATA[1884,17] := 1.0;
   DATA[1884,18] := 1.0;
   DATA[1884,19] := 2.0;
   DATA[1884,20] := 148.808;
   DATA[1884,21] := 154.7552;
   DATA[1884,22] := 1.716721;
   DATA[1884,23] := 820.1743;
   DATA[1884,24] := 2.0;
   DATA[1884,25] := 2.0;
   DATA[1884,26] := 7.874135;
   DATA[1884,27] := 143.6811;
   DATA[1884,28] := 262.3366;
   DATA[1884,29] := 12.03538;
   DATA[1884,30] := 1.724942;
   DATA[1884,31] := 1.264634;
   DATA[1884,32] := 0.7355248;
   DATA[1884,33] := 0.3084265;
   DATA[1884,34] := 2.0;
   DATA[1884,35] := 249.984;
   DATA[1884,36] := 1.762086;
   DATA[1884,37] := 188.8939;
   DATA[1884,38] := 0.000128152;
   DATA[1884,39] := 1.0;
   DATA[1884,40] := 1.0;
   DATA[1885,0] := 2.539154;
   DATA[1885,1] := 859.0466;
   DATA[1885,2] := 2.0;
   DATA[1885,3] := 2.0;
   DATA[1885,4] := 262.6891;
   DATA[1885,5] := 8.39163;
   DATA[1885,6] := 332.9659;
   DATA[1885,7] := 2.463589;
   DATA[1885,8] := 2.0;
   DATA[1885,9] := 2.0;
   DATA[1885,10] := 2.0;
   DATA[1885,11] := 19.72598;
   DATA[1885,12] := 2.207091;
   DATA[1885,13] := 791.9844;
   DATA[1885,14] := 1.0;
   DATA[1885,15] := 2.0;
   DATA[1885,16] := 1.0;
   DATA[1885,17] := 1.0;
   DATA[1885,18] := 1.0;
   DATA[1885,19] := 2.0;
   DATA[1885,20] := 148.808;
   DATA[1885,21] := 154.7552;
   DATA[1885,22] := 1.716721;
   DATA[1885,23] := 820.4435;
   DATA[1885,24] := 2.0;
   DATA[1885,25] := 2.0;
   DATA[1885,26] := 7.874135;
   DATA[1885,27] := 143.6811;
   DATA[1885,28] := 262.3366;
   DATA[1885,29] := 12.03538;
   DATA[1885,30] := 1.724942;
   DATA[1885,31] := 1.255924;
   DATA[1885,32] := 0.7355248;
   DATA[1885,33] := 0.3084265;
   DATA[1885,34] := 2.0;
   DATA[1885,35] := 249.984;
   DATA[1885,36] := 1.762086;
   DATA[1885,37] := 188.8939;
   DATA[1885,38] := 0.000128152;
   DATA[1885,39] := 1.0;
   DATA[1885,40] := 1.0;
   DATA[1886,0] := 2.579188;
   DATA[1886,1] := 858.7719;
   DATA[1886,2] := 2.0;
   DATA[1886,3] := 2.0;
   DATA[1886,4] := 262.6891;
   DATA[1886,5] := 8.390669;
   DATA[1886,6] := 332.8377;
   DATA[1886,7] := 2.463589;
   DATA[1886,8] := 2.0;
   DATA[1886,9] := 2.0;
   DATA[1886,10] := 2.0;
   DATA[1886,11] := 19.63634;
   DATA[1886,12] := 2.207091;
   DATA[1886,13] := 791.7842;
   DATA[1886,14] := 1.0;
   DATA[1886,15] := 2.0;
   DATA[1886,16] := 1.0;
   DATA[1886,17] := 1.0;
   DATA[1886,18] := 1.0;
   DATA[1886,19] := 2.0;
   DATA[1886,20] := 148.808;
   DATA[1886,21] := 154.7552;
   DATA[1886,22] := 1.714542;
   DATA[1886,23] := 820.5973;
   DATA[1886,24] := 2.0;
   DATA[1886,25] := 2.0;
   DATA[1886,26] := 7.874135;
   DATA[1886,27] := 143.6811;
   DATA[1886,28] := 262.3366;
   DATA[1886,29] := 12.03538;
   DATA[1886,30] := 1.724942;
   DATA[1886,31] := 1.269502;
   DATA[1886,32] := 0.7352687;
   DATA[1886,33] := 0.3084265;
   DATA[1886,34] := 2.0;
   DATA[1886,35] := 249.984;
   DATA[1886,36] := 1.762086;
   DATA[1886,37] := 188.8939;
   DATA[1886,38] := 0.000128152;
   DATA[1886,39] := 1.0;
   DATA[1886,40] := 1.0;
   DATA[1887,0] := 2.618903;
   DATA[1887,1] := 858.7326;
   DATA[1887,2] := 2.0;
   DATA[1887,3] := 2.0;
   DATA[1887,4] := 262.6891;
   DATA[1887,5] := 8.390669;
   DATA[1887,6] := 332.8377;
   DATA[1887,7] := 2.463589;
   DATA[1887,8] := 2.0;
   DATA[1887,9] := 2.0;
   DATA[1887,10] := 2.0;
   DATA[1887,11] := 19.63634;
   DATA[1887,12] := 2.209269;
   DATA[1887,13] := 791.5438;
   DATA[1887,14] := 1.0;
   DATA[1887,15] := 2.0;
   DATA[1887,16] := 1.0;
   DATA[1887,17] := 1.0;
   DATA[1887,18] := 1.0;
   DATA[1887,19] := 2.0;
   DATA[1887,20] := 148.808;
   DATA[1887,21] := 154.7552;
   DATA[1887,22] := 1.714542;
   DATA[1887,23] := 820.7896;
   DATA[1887,24] := 2.0;
   DATA[1887,25] := 2.0;
   DATA[1887,26] := 7.874135;
   DATA[1887,27] := 143.6811;
   DATA[1887,28] := 262.3366;
   DATA[1887,29] := 12.03538;
   DATA[1887,30] := 1.72443;
   DATA[1887,31] := 1.281286;
   DATA[1887,32] := 0.7352687;
   DATA[1887,33] := 0.3084265;
   DATA[1887,34] := 2.0;
   DATA[1887,35] := 249.984;
   DATA[1887,36] := 1.762086;
   DATA[1887,37] := 188.8939;
   DATA[1887,38] := 0.000128152;
   DATA[1887,39] := 1.0;
   DATA[1887,40] := 1.0;
   DATA[1888,0] := 2.649649;
   DATA[1888,1] := 858.4971;
   DATA[1888,2] := 2.0;
   DATA[1888,3] := 2.0;
   DATA[1888,4] := 262.6891;
   DATA[1888,5] := 8.390669;
   DATA[1888,6] := 332.8377;
   DATA[1888,7] := 2.463589;
   DATA[1888,8] := 2.0;
   DATA[1888,9] := 2.0;
   DATA[1888,10] := 2.0;
   DATA[1888,11] := 19.62033;
   DATA[1888,12] := 2.210166;
   DATA[1888,13] := 791.3837;
   DATA[1888,14] := 1.0;
   DATA[1888,15] := 2.0;
   DATA[1888,16] := 1.0;
   DATA[1888,17] := 1.0;
   DATA[1888,18] := 1.0;
   DATA[1888,19] := 2.0;
   DATA[1888,20] := 148.808;
   DATA[1888,21] := 154.7552;
   DATA[1888,22] := 1.714542;
   DATA[1888,23] := 820.7511;
   DATA[1888,24] := 2.0;
   DATA[1888,25] := 2.0;
   DATA[1888,26] := 7.874135;
   DATA[1888,27] := 143.5529;
   DATA[1888,28] := 262.3366;
   DATA[1888,29] := 12.03538;
   DATA[1888,30] := 1.72443;
   DATA[1888,31] := 1.287434;
   DATA[1888,32] := 0.7352687;
   DATA[1888,33] := 0.3084265;
   DATA[1888,34] := 2.0;
   DATA[1888,35] := 249.984;
   DATA[1888,36] := 1.762086;
   DATA[1888,37] := 188.8939;
   DATA[1888,38] := 0.000128152;
   DATA[1888,39] := 1.0;
   DATA[1888,40] := 1.0;
   DATA[1889,0] := 2.659578;
   DATA[1889,1] := 858.7719;
   DATA[1889,2] := 2.0;
   DATA[1889,3] := 2.0;
   DATA[1889,4] := 262.6891;
   DATA[1889,5] := 8.390669;
   DATA[1889,6] := 333.0172;
   DATA[1889,7] := 2.463589;
   DATA[1889,8] := 2.0;
   DATA[1889,9] := 2.0;
   DATA[1889,10] := 2.0;
   DATA[1889,11] := 19.62033;
   DATA[1889,12] := 2.210166;
   DATA[1889,13] := 791.7842;
   DATA[1889,14] := 1.0;
   DATA[1889,15] := 2.0;
   DATA[1889,16] := 1.0;
   DATA[1889,17] := 1.0;
   DATA[1889,18] := 1.0;
   DATA[1889,19] := 2.0;
   DATA[1889,20] := 148.808;
   DATA[1889,21] := 154.7552;
   DATA[1889,22] := 1.714542;
   DATA[1889,23] := 821.1356;
   DATA[1889,24] := 2.0;
   DATA[1889,25] := 2.0;
   DATA[1889,26] := 7.874135;
   DATA[1889,27] := 143.5529;
   DATA[1889,28] := 262.3366;
   DATA[1889,29] := 12.03538;
   DATA[1889,30] := 1.72443;
   DATA[1889,31] := 1.292174;
   DATA[1889,32] := 0.7352687;
   DATA[1889,33] := 0.3084265;
   DATA[1889,34] := 2.0;
   DATA[1889,35] := 249.984;
   DATA[1889,36] := 1.762086;
   DATA[1889,37] := 188.8939;
   DATA[1889,38] := 0.000128152;
   DATA[1889,39] := 1.0;
   DATA[1889,40] := 1.0;
   DATA[1890,0] := 2.663421;
   DATA[1890,1] := 858.7326;
   DATA[1890,2] := 2.0;
   DATA[1890,3] := 2.0;
   DATA[1890,4] := 262.6891;
   DATA[1890,5] := 8.390669;
   DATA[1890,6] := 333.0172;
   DATA[1890,7] := 2.466536;
   DATA[1890,8] := 2.0;
   DATA[1890,9] := 2.0;
   DATA[1890,10] := 2.0;
   DATA[1890,11] := 19.68436;
   DATA[1890,12] := 2.212215;
   DATA[1890,13] := 791.7441;
   DATA[1890,14] := 1.0;
   DATA[1890,15] := 2.0;
   DATA[1890,16] := 1.0;
   DATA[1890,17] := 1.0;
   DATA[1890,18] := 1.0;
   DATA[1890,19] := 2.0;
   DATA[1890,20] := 148.808;
   DATA[1890,21] := 154.7552;
   DATA[1890,22] := 1.712107;
   DATA[1890,23] := 820.7896;
   DATA[1890,24] := 2.0;
   DATA[1890,25] := 2.0;
   DATA[1890,26] := 7.874135;
   DATA[1890,27] := 143.5529;
   DATA[1890,28] := 262.3366;
   DATA[1890,29] := 12.03538;
   DATA[1890,30] := 1.72443;
   DATA[1890,31] := 1.299219;
   DATA[1890,32] := 0.7352687;
   DATA[1890,33] := 0.3084265;
   DATA[1890,34] := 2.0;
   DATA[1890,35] := 249.984;
   DATA[1890,36] := 1.762086;
   DATA[1890,37] := 188.8939;
   DATA[1890,38] := 0.000128152;
   DATA[1890,39] := 1.0;
   DATA[1890,40] := 1.0;
   DATA[1891,0] := 2.640361;
   DATA[1891,1] := 858.9288;
   DATA[1891,2] := 2.0;
   DATA[1891,3] := 2.0;
   DATA[1891,4] := 262.5609;
   DATA[1891,5] := 8.390669;
   DATA[1891,6] := 333.0172;
   DATA[1891,7] := 2.467433;
   DATA[1891,8] := 2.0;
   DATA[1891,9] := 2.0;
   DATA[1891,10] := 2.0;
   DATA[1891,11] := 19.71637;
   DATA[1891,12] := 2.2126;
   DATA[1891,13] := 792.0646;
   DATA[1891,14] := 1.0;
   DATA[1891,15] := 2.0;
   DATA[1891,16] := 1.0;
   DATA[1891,17] := 1.0;
   DATA[1891,18] := 1.0;
   DATA[1891,19] := 2.0;
   DATA[1891,20] := 148.808;
   DATA[1891,21] := 154.7552;
   DATA[1891,22] := 1.712107;
   DATA[1891,23] := 821.0203;
   DATA[1891,24] := 2.0;
   DATA[1891,25] := 2.0;
   DATA[1891,26] := 7.874135;
   DATA[1891,27] := 143.5529;
   DATA[1891,28] := 262.3366;
   DATA[1891,29] := 12.03538;
   DATA[1891,30] := 1.72507;
   DATA[1891,31] := 1.302165;
   DATA[1891,32] := 0.7352687;
   DATA[1891,33] := 0.3084265;
   DATA[1891,34] := 2.0;
   DATA[1891,35] := 249.984;
   DATA[1891,36] := 1.730048;
   DATA[1891,37] := 188.8939;
   DATA[1891,38] := 0.000128152;
   DATA[1891,39] := 1.0;
   DATA[1891,40] := 1.0;
   DATA[1892,0] := 2.640361;
   DATA[1892,1] := 858.9288;
   DATA[1892,2] := 2.0;
   DATA[1892,3] := 2.0;
   DATA[1892,4] := 262.5609;
   DATA[1892,5] := 8.390669;
   DATA[1892,6] := 333.0172;
   DATA[1892,7] := 2.467433;
   DATA[1892,8] := 2.0;
   DATA[1892,9] := 2.0;
   DATA[1892,10] := 2.0;
   DATA[1892,11] := 19.71637;
   DATA[1892,12] := 2.2126;
   DATA[1892,13] := 792.0646;
   DATA[1892,14] := 1.0;
   DATA[1892,15] := 2.0;
   DATA[1892,16] := 1.0;
   DATA[1892,17] := 1.0;
   DATA[1892,18] := 1.0;
   DATA[1892,19] := 2.0;
   DATA[1892,20] := 148.808;
   DATA[1892,21] := 154.7552;
   DATA[1892,22] := 1.712107;
   DATA[1892,23] := 821.0203;
   DATA[1892,24] := 2.0;
   DATA[1892,25] := 2.0;
   DATA[1892,26] := 7.874135;
   DATA[1892,27] := 143.5529;
   DATA[1892,28] := 262.3366;
   DATA[1892,29] := 12.03538;
   DATA[1892,30] := 1.72507;
   DATA[1892,31] := 1.302165;
   DATA[1892,32] := 0.7352687;
   DATA[1892,33] := 0.3084265;
   DATA[1892,34] := 2.0;
   DATA[1892,35] := 249.984;
   DATA[1892,36] := 1.730048;
   DATA[1892,37] := 188.8939;
   DATA[1892,38] := 0.000128152;
   DATA[1892,39] := 1.0;
   DATA[1892,40] := 1.0;
   DATA[1893,0] := 2.623387;
   DATA[1893,1] := 859.7139;
   DATA[1893,2] := 2.0;
   DATA[1893,3] := 2.0;
   DATA[1893,4] := 262.5609;
   DATA[1893,5] := 8.390669;
   DATA[1893,6] := 332.9659;
   DATA[1893,7] := 2.46769;
   DATA[1893,8] := 2.0;
   DATA[1893,9] := 2.0;
   DATA[1893,10] := 2.0;
   DATA[1893,11] := 19.71637;
   DATA[1893,12] := 2.2126;
   DATA[1893,13] := 792.3049;
   DATA[1893,14] := 1.0;
   DATA[1893,15] := 2.0;
   DATA[1893,16] := 1.0;
   DATA[1893,17] := 1.0;
   DATA[1893,18] := 1.0;
   DATA[1893,19] := 2.0;
   DATA[1893,20] := 148.808;
   DATA[1893,21] := 154.7552;
   DATA[1893,22] := 1.712107;
   DATA[1893,23] := 820.9049;
   DATA[1893,24] := 2.0;
   DATA[1893,25] := 2.0;
   DATA[1893,26] := 7.874135;
   DATA[1893,27] := 143.5529;
   DATA[1893,28] := 262.1764;
   DATA[1893,29] := 12.03538;
   DATA[1893,30] := 1.72507;
   DATA[1893,31] := 1.302165;
   DATA[1893,32] := 0.7352687;
   DATA[1893,33] := 0.3084265;
   DATA[1893,34] := 2.0;
   DATA[1893,35] := 249.984;
   DATA[1893,36] := 1.730048;
   DATA[1893,37] := 188.8939;
   DATA[1893,38] := 0.000128152;
   DATA[1893,39] := 1.0;
   DATA[1893,40] := 1.0;
   DATA[1894,0] := 2.623387;
   DATA[1894,1] := 859.6747;
   DATA[1894,2] := 2.0;
   DATA[1894,3] := 2.0;
   DATA[1894,4] := 262.5609;
   DATA[1894,5] := 8.390669;
   DATA[1894,6] := 332.8634;
   DATA[1894,7] := 2.46769;
   DATA[1894,8] := 2.0;
   DATA[1894,9] := 2.0;
   DATA[1894,10] := 2.0;
   DATA[1894,11] := 19.72277;
   DATA[1894,12] := 2.2126;
   DATA[1894,13] := 792.3049;
   DATA[1894,14] := 1.0;
   DATA[1894,15] := 2.0;
   DATA[1894,16] := 1.0;
   DATA[1894,17] := 1.0;
   DATA[1894,18] := 1.0;
   DATA[1894,19] := 2.0;
   DATA[1894,20] := 148.808;
   DATA[1894,21] := 154.7552;
   DATA[1894,22] := 1.712107;
   DATA[1894,23] := 821.597;
   DATA[1894,24] := 2.0;
   DATA[1894,25] := 2.0;
   DATA[1894,26] := 7.874135;
   DATA[1894,27] := 143.5529;
   DATA[1894,28] := 262.1764;
   DATA[1894,29] := 12.03538;
   DATA[1894,30] := 1.72507;
   DATA[1894,31] := 1.281542;
   DATA[1894,32] := 0.7352687;
   DATA[1894,33] := 0.3084265;
   DATA[1894,34] := 2.0;
   DATA[1894,35] := 249.984;
   DATA[1894,36] := 1.730048;
   DATA[1894,37] := 188.8939;
   DATA[1894,38] := 0.000128152;
   DATA[1894,39] := 1.0;
   DATA[1894,40] := 1.0;
   DATA[1895,0] := 2.619223;
   DATA[1895,1] := 860.1457;
   DATA[1895,2] := 2.0;
   DATA[1895,3] := 2.0;
   DATA[1895,4] := 262.5609;
   DATA[1895,5] := 8.390669;
   DATA[1895,6] := 332.8634;
   DATA[1895,7] := 2.46769;
   DATA[1895,8] := 2.0;
   DATA[1895,9] := 2.0;
   DATA[1895,10] := 2.0;
   DATA[1895,11] := 19.72277;
   DATA[1895,12] := 2.211575;
   DATA[1895,13] := 792.5853;
   DATA[1895,14] := 1.0;
   DATA[1895,15] := 2.0;
   DATA[1895,16] := 1.0;
   DATA[1895,17] := 1.0;
   DATA[1895,18] := 1.0;
   DATA[1895,19] := 2.0;
   DATA[1895,20] := 148.808;
   DATA[1895,21] := 154.7552;
   DATA[1895,22] := 1.712107;
   DATA[1895,23] := 821.4817;
   DATA[1895,24] := 2.0;
   DATA[1895,25] := 2.0;
   DATA[1895,26] := 7.874135;
   DATA[1895,27] := 143.5529;
   DATA[1895,28] := 262.1764;
   DATA[1895,29] := 12.03538;
   DATA[1895,30] := 1.72507;
   DATA[1895,31] := 1.271423;
   DATA[1895,32] := 0.7352687;
   DATA[1895,33] := 0.3084265;
   DATA[1895,34] := 2.0;
   DATA[1895,35] := 250.0801;
   DATA[1895,36] := 1.730048;
   DATA[1895,37] := 188.8939;
   DATA[1895,38] := 0.000128152;
   DATA[1895,39] := 1.0;
   DATA[1895,40] := 1.0;
   DATA[1896,0] := 2.60481;
   DATA[1896,1] := 859.9494;
   DATA[1896,2] := 2.0;
   DATA[1896,3] := 2.0;
   DATA[1896,4] := 262.5609;
   DATA[1896,5] := 8.390669;
   DATA[1896,6] := 332.8634;
   DATA[1896,7] := 2.4691;
   DATA[1896,8] := 2.0;
   DATA[1896,9] := 2.0;
   DATA[1896,10] := 2.0;
   DATA[1896,11] := 19.72277;
   DATA[1896,12] := 2.210294;
   DATA[1896,13] := 792.5452;
   DATA[1896,14] := 1.0;
   DATA[1896,15] := 2.0;
   DATA[1896,16] := 1.0;
   DATA[1896,17] := 1.0;
   DATA[1896,18] := 1.0;
   DATA[1896,19] := 2.0;
   DATA[1896,20] := 148.808;
   DATA[1896,21] := 154.7552;
   DATA[1896,22] := 1.712107;
   DATA[1896,23] := 821.7509;
   DATA[1896,24] := 2.0;
   DATA[1896,25] := 2.0;
   DATA[1896,26] := 7.874135;
   DATA[1896,27] := 143.5529;
   DATA[1896,28] := 262.1764;
   DATA[1896,29] := 12.30454;
   DATA[1896,30] := 1.72507;
   DATA[1896,31] := 1.271423;
   DATA[1896,32] := 0.7371892;
   DATA[1896,33] := 0.3084265;
   DATA[1896,34] := 2.0;
   DATA[1896,35] := 250.3525;
   DATA[1896,36] := 1.730048;
   DATA[1896,37] := 189.1342;
   DATA[1896,38] := 0.000128152;
   DATA[1896,39] := 1.0;
   DATA[1896,40] := 1.0;
   DATA[1897,0] := 2.579188;
   DATA[1897,1] := 860.4597;
   DATA[1897,2] := 2.0;
   DATA[1897,3] := 2.0;
   DATA[1897,4] := 262.5609;
   DATA[1897,5] := 8.390669;
   DATA[1897,6] := 332.8634;
   DATA[1897,7] := 2.4691;
   DATA[1897,8] := 2.0;
   DATA[1897,9] := 2.0;
   DATA[1897,10] := 2.0;
   DATA[1897,11] := 19.72277;
   DATA[1897,12] := 2.210037;
   DATA[1897,13] := 792.5452;
   DATA[1897,14] := 1.0;
   DATA[1897,15] := 2.0;
   DATA[1897,16] := 1.0;
   DATA[1897,17] := 1.0;
   DATA[1897,18] := 1.0;
   DATA[1897,19] := 2.0;
   DATA[1897,20] := 148.808;
   DATA[1897,21] := 154.7552;
   DATA[1897,22] := 1.714029;
   DATA[1897,23] := 821.3663;
   DATA[1897,24] := 2.0;
   DATA[1897,25] := 2.0;
   DATA[1897,26] := 7.874135;
   DATA[1897,27] := 143.5529;
   DATA[1897,28] := 262.1764;
   DATA[1897,29] := 12.30454;
   DATA[1897,30] := 1.72507;
   DATA[1897,31] := 1.271423;
   DATA[1897,32] := 0.7377012;
   DATA[1897,33] := 0.3084265;
   DATA[1897,34] := 2.0;
   DATA[1897,35] := 250.3525;
   DATA[1897,36] := 1.730048;
   DATA[1897,37] := 189.1823;
   DATA[1897,38] := 0.000128152;
   DATA[1897,39] := 1.0;
   DATA[1897,40] := 1.0;
   DATA[1898,0] := 2.567979;
   DATA[1898,1] := 860.6559;
   DATA[1898,2] := 2.0;
   DATA[1898,3] := 2.0;
   DATA[1898,4] := 262.5609;
   DATA[1898,5] := 8.390669;
   DATA[1898,6] := 332.8634;
   DATA[1898,7] := 2.4691;
   DATA[1898,8] := 2.0;
   DATA[1898,9] := 2.0;
   DATA[1898,10] := 2.0;
   DATA[1898,11] := 19.72598;
   DATA[1898,12] := 2.207731;
   DATA[1898,13] := 792.9457;
   DATA[1898,14] := 1.0;
   DATA[1898,15] := 2.0;
   DATA[1898,16] := 1.0;
   DATA[1898,17] := 1.0;
   DATA[1898,18] := 1.0;
   DATA[1898,19] := 2.0;
   DATA[1898,20] := 148.808;
   DATA[1898,21] := 154.7552;
   DATA[1898,22] := 1.716464;
   DATA[1898,23] := 821.4817;
   DATA[1898,24] := 2.0;
   DATA[1898,25] := 2.0;
   DATA[1898,26] := 7.874135;
   DATA[1898,27] := 143.5529;
   DATA[1898,28] := 262.1764;
   DATA[1898,29] := 12.03538;
   DATA[1898,30] := 1.725455;
   DATA[1898,31] := 1.271423;
   DATA[1898,32] := 0.7370611;
   DATA[1898,33] := 0.3084265;
   DATA[1898,34] := 2.0;
   DATA[1898,35] := 250.3525;
   DATA[1898,36] := 1.730048;
   DATA[1898,37] := 189.1823;
   DATA[1898,38] := 0.000128152;
   DATA[1898,39] := 1.0;
   DATA[1898,40] := 1.0;
   DATA[1899,0] := 2.545559;
   DATA[1899,1] := 860.2242;
   DATA[1899,2] := 2.0;
   DATA[1899,3] := 2.0;
   DATA[1899,4] := 262.5609;
   DATA[1899,5] := 8.392271;
   DATA[1899,6] := 332.8634;
   DATA[1899,7] := 2.467946;
   DATA[1899,8] := 2.0;
   DATA[1899,9] := 2.0;
   DATA[1899,10] := 2.0;
   DATA[1899,11] := 19.72598;
   DATA[1899,12] := 2.207347;
   DATA[1899,13] := 792.7054;
   DATA[1899,14] := 1.0;
   DATA[1899,15] := 2.0;
   DATA[1899,16] := 1.0;
   DATA[1899,17] := 1.0;
   DATA[1899,18] := 1.0;
   DATA[1899,19] := 2.0;
   DATA[1899,20] := 148.808;
   DATA[1899,21] := 154.7552;
   DATA[1899,22] := 1.716464;
   DATA[1899,23] := 821.1356;
   DATA[1899,24] := 2.0;
   DATA[1899,25] := 2.0;
   DATA[1899,26] := 7.874135;
   DATA[1899,27] := 143.6042;
   DATA[1899,28] := 262.1764;
   DATA[1899,29] := 12.03538;
   DATA[1899,30] := 1.726352;
   DATA[1899,31] := 1.268477;
   DATA[1899,32] := 0.7370611;
   DATA[1899,33] := 0.3084265;
   DATA[1899,34] := 2.0;
   DATA[1899,35] := 250.3525;
   DATA[1899,36] := 1.730048;
   DATA[1899,37] := 189.1823;
   DATA[1899,38] := 0.000128152;
   DATA[1899,39] := 1.0;
   DATA[1899,40] := 1.0;
   DATA[1900,0] := 2.538513;
   DATA[1900,1] := 860.2634;
   DATA[1900,2] := 2.0;
   DATA[1900,3] := 2.0;
   DATA[1900,4] := 262.5609;
   DATA[1900,5] := 8.392271;
   DATA[1900,6] := 332.7096;
   DATA[1900,7] := 2.466408;
   DATA[1900,8] := 2.0;
   DATA[1900,9] := 2.0;
   DATA[1900,10] := 2.0;
   DATA[1900,11] := 19.72598;
   DATA[1900,12] := 2.206835;
   DATA[1900,13] := 793.0659;
   DATA[1900,14] := 1.0;
   DATA[1900,15] := 2.0;
   DATA[1900,16] := 1.0;
   DATA[1900,17] := 1.0;
   DATA[1900,18] := 1.0;
   DATA[1900,19] := 2.0;
   DATA[1900,20] := 148.808;
   DATA[1900,21] := 154.7552;
   DATA[1900,22] := 1.716464;
   DATA[1900,23] := 820.9434;
   DATA[1900,24] := 2.0;
   DATA[1900,25] := 2.0;
   DATA[1900,26] := 7.874135;
   DATA[1900,27] := 143.6042;
   DATA[1900,28] := 262.3045;
   DATA[1900,29] := 12.03538;
   DATA[1900,30] := 1.728788;
   DATA[1900,31] := 1.264891;
   DATA[1900,32] := 0.7370611;
   DATA[1900,33] := 0.306761;
   DATA[1900,34] := 2.0;
   DATA[1900,35] := 250.3525;
   DATA[1900,36] := 1.730048;
   DATA[1900,37] := 189.1823;
   DATA[1900,38] := 0.000128152;
   DATA[1900,39] := 1.0;
   DATA[1900,40] := 1.0;
   DATA[1901,0] := 2.514813;
   DATA[1901,1] := 860.4597;
   DATA[1901,2] := 2.0;
   DATA[1901,3] := 2.0;
   DATA[1901,4] := 262.5609;
   DATA[1901,5] := 8.393232;
   DATA[1901,6] := 332.7096;
   DATA[1901,7] := 2.466408;
   DATA[1901,8] := 2.0;
   DATA[1901,9] := 2.0;
   DATA[1901,10] := 2.0;
   DATA[1901,11] := 19.72277;
   DATA[1901,12] := 2.207731;
   DATA[1901,13] := 792.9858;
   DATA[1901,14] := 1.0;
   DATA[1901,15] := 2.0;
   DATA[1901,16] := 1.0;
   DATA[1901,17] := 1.0;
   DATA[1901,18] := 1.0;
   DATA[1901,19] := 2.0;
   DATA[1901,20] := 148.808;
   DATA[1901,21] := 154.7552;
   DATA[1901,22] := 1.716464;
   DATA[1901,23] := 821.0203;
   DATA[1901,24] := 2.0;
   DATA[1901,25] := 2.0;
   DATA[1901,26] := 7.874135;
   DATA[1901,27] := 143.6042;
   DATA[1901,28] := 262.4968;
   DATA[1901,29] := 12.03538;
   DATA[1901,30] := 1.728788;
   DATA[1901,31] := 1.279877;
   DATA[1901,32] := 0.7370611;
   DATA[1901,33] := 0.3066329;
   DATA[1901,34] := 2.0;
   DATA[1901,35] := 250.3525;
   DATA[1901,36] := 1.730048;
   DATA[1901,37] := 189.1823;
   DATA[1901,38] := 0.000128152;
   DATA[1901,39] := 1.0;
   DATA[1901,40] := 1.0;
   DATA[1902,0] := 2.508087;
   DATA[1902,1] := 860.342;
   DATA[1902,2] := 2.0;
   DATA[1902,3] := 2.0;
   DATA[1902,4] := 262.5609;
   DATA[1902,5] := 8.393232;
   DATA[1902,6] := 332.7096;
   DATA[1902,7] := 2.466408;
   DATA[1902,8] := 2.0;
   DATA[1902,9] := 2.0;
   DATA[1902,10] := 2.0;
   DATA[1902,11] := 19.72277;
   DATA[1902,12] := 2.210294;
   DATA[1902,13] := 793.106;
   DATA[1902,14] := 1.0;
   DATA[1902,15] := 2.0;
   DATA[1902,16] := 1.0;
   DATA[1902,17] := 1.0;
   DATA[1902,18] := 1.0;
   DATA[1902,19] := 2.0;
   DATA[1902,20] := 148.808;
   DATA[1902,21] := 154.7552;
   DATA[1902,22] := 1.716721;
   DATA[1902,23] := 820.6357;
   DATA[1902,24] := 2.0;
   DATA[1902,25] := 2.0;
   DATA[1902,26] := 7.874135;
   DATA[1902,27] := 143.6042;
   DATA[1902,28] := 262.4968;
   DATA[1902,29] := 12.03538;
   DATA[1902,30] := 1.727634;
   DATA[1902,31] := 1.280902;
   DATA[1902,32] := 0.7348846;
   DATA[1902,33] := 0.3066329;
   DATA[1902,34] := 2.0;
   DATA[1902,35] := 250.3525;
   DATA[1902,36] := 1.730048;
   DATA[1902,37] := 189.1823;
   DATA[1902,38] := 0.000128152;
   DATA[1902,39] := 1.0;
   DATA[1902,40] := 1.0;
   DATA[1903,0] := 2.491432;
   DATA[1903,1] := 860.1064;
   DATA[1903,2] := 2.0;
   DATA[1903,3] := 2.0;
   DATA[1903,4] := 262.5609;
   DATA[1903,5] := 8.393232;
   DATA[1903,6] := 332.5814;
   DATA[1903,7] := 2.466408;
   DATA[1903,8] := 2.0;
   DATA[1903,9] := 2.0;
   DATA[1903,10] := 2.0;
   DATA[1903,11] := 19.72277;
   DATA[1903,12] := 2.210294;
   DATA[1903,13] := 793.3463;
   DATA[1903,14] := 1.0;
   DATA[1903,15] := 2.0;
   DATA[1903,16] := 1.0;
   DATA[1903,17] := 1.0;
   DATA[1903,18] := 1.0;
   DATA[1903,19] := 2.0;
   DATA[1903,20] := 148.808;
   DATA[1903,21] := 154.7808;
   DATA[1903,22] := 1.716721;
   DATA[1903,23] := 820.3281;
   DATA[1903,24] := 2.0;
   DATA[1903,25] := 2.0;
   DATA[1903,26] := 7.874135;
   DATA[1903,27] := 143.6042;
   DATA[1903,28] := 262.4968;
   DATA[1903,29] := 12.03538;
   DATA[1903,30] := 1.72507;
   DATA[1903,31] := 1.276547;
   DATA[1903,32] := 0.7348846;
   DATA[1903,33] := 0.3075937;
   DATA[1903,34] := 2.0;
   DATA[1903,35] := 250.3525;
   DATA[1903,36] := 1.730048;
   DATA[1903,37] := 189.1823;
   DATA[1903,38] := 0.000128152;
   DATA[1903,39] := 1.0;
   DATA[1903,40] := 1.0;
   DATA[1904,0] := 2.476059;
   DATA[1904,1] := 859.9102;
   DATA[1904,2] := 2.0;
   DATA[1904,3] := 2.0;
   DATA[1904,4] := 262.5609;
   DATA[1904,5] := 8.393232;
   DATA[1904,6] := 332.5814;
   DATA[1904,7] := 2.466024;
   DATA[1904,8] := 2.0;
   DATA[1904,9] := 2.0;
   DATA[1904,10] := 2.0;
   DATA[1904,11] := 19.72277;
   DATA[1904,12] := 2.210294;
   DATA[1904,13] := 793.7068;
   DATA[1904,14] := 1.0;
   DATA[1904,15] := 2.0;
   DATA[1904,16] := 1.0;
   DATA[1904,17] := 1.0;
   DATA[1904,18] := 1.0;
   DATA[1904,19] := 2.0;
   DATA[1904,20] := 148.808;
   DATA[1904,21] := 154.7808;
   DATA[1904,22] := 1.716721;
   DATA[1904,23] := 819.7898;
   DATA[1904,24] := 2.0;
   DATA[1904,25] := 2.0;
   DATA[1904,26] := 7.874135;
   DATA[1904,27] := 143.6042;
   DATA[1904,28] := 262.3045;
   DATA[1904,29] := 12.03538;
   DATA[1904,30] := 1.72507;
   DATA[1904,31] := 1.290765;
   DATA[1904,32] := 0.7348846;
   DATA[1904,33] := 0.3084265;
   DATA[1904,34] := 2.0;
   DATA[1904,35] := 250.3525;
   DATA[1904,36] := 1.730048;
   DATA[1904,37] := 189.1823;
   DATA[1904,38] := 0.000128152;
   DATA[1904,39] := 1.0;
   DATA[1904,40] := 1.0;
   DATA[1905,0] := 2.458764;
   DATA[1905,1] := 860.028;
   DATA[1905,2] := 2.0;
   DATA[1905,3] := 2.0;
   DATA[1905,4] := 262.5609;
   DATA[1905,5] := 8.390669;
   DATA[1905,6] := 332.5814;
   DATA[1905,7] := 2.463461;
   DATA[1905,8] := 2.0;
   DATA[1905,9] := 2.0;
   DATA[1905,10] := 2.0;
   DATA[1905,11] := 19.72277;
   DATA[1905,12] := 2.211959;
   DATA[1905,13] := 793.867;
   DATA[1905,14] := 1.0;
   DATA[1905,15] := 2.0;
   DATA[1905,16] := 1.0;
   DATA[1905,17] := 1.0;
   DATA[1905,18] := 1.0;
   DATA[1905,19] := 2.0;
   DATA[1905,20] := 148.808;
   DATA[1905,21] := 154.7808;
   DATA[1905,22] := 1.714158;
   DATA[1905,23] := 819.4437;
   DATA[1905,24] := 2.0;
   DATA[1905,25] := 2.0;
   DATA[1905,26] := 7.874135;
   DATA[1905,27] := 143.6042;
   DATA[1905,28] := 262.3045;
   DATA[1905,29] := 12.03538;
   DATA[1905,30] := 1.72507;
   DATA[1905,31] := 1.292046;
   DATA[1905,32] := 0.7348846;
   DATA[1905,33] := 0.3084265;
   DATA[1905,34] := 2.0;
   DATA[1905,35] := 250.3525;
   DATA[1905,36] := 1.730048;
   DATA[1905,37] := 189.1823;
   DATA[1905,38] := 0.000128152;
   DATA[1905,39] := 1.0;
   DATA[1905,40] := 1.0;
   DATA[1906,0] := 2.447234;
   DATA[1906,1] := 860.2242;
   DATA[1906,2] := 2.0;
   DATA[1906,3] := 2.0;
   DATA[1906,4] := 262.5609;
   DATA[1906,5] := 8.390669;
   DATA[1906,6] := 332.5814;
   DATA[1906,7] := 2.463461;
   DATA[1906,8] := 2.0;
   DATA[1906,9] := 2.0;
   DATA[1906,10] := 2.0;
   DATA[1906,11] := 19.76759;
   DATA[1906,12] := 2.212215;
   DATA[1906,13] := 793.5065;
   DATA[1906,14] := 1.0;
   DATA[1906,15] := 2.0;
   DATA[1906,16] := 1.0;
   DATA[1906,17] := 1.0;
   DATA[1906,18] := 1.0;
   DATA[1906,19] := 2.0;
   DATA[1906,20] := 148.808;
   DATA[1906,21] := 154.7808;
   DATA[1906,22] := 1.713389;
   DATA[1906,23] := 819.6744;
   DATA[1906,24] := 2.0;
   DATA[1906,25] := 2.0;
   DATA[1906,26] := 7.874135;
   DATA[1906,27] := 143.6042;
   DATA[1906,28] := 262.3045;
   DATA[1906,29] := 12.22763;
   DATA[1906,30] := 1.726737;
   DATA[1906,31] := 1.306136;
   DATA[1906,32] := 0.7348846;
   DATA[1906,33] := 0.3084265;
   DATA[1906,34] := 2.0;
   DATA[1906,35] := 250.3525;
   DATA[1906,36] := 1.730048;
   DATA[1906,37] := 189.1823;
   DATA[1906,38] := 0.000128152;
   DATA[1906,39] := 1.0;
   DATA[1906,40] := 1.0;
   DATA[1907,0] := 2.433783;
   DATA[1907,1] := 859.8317;
   DATA[1907,2] := 2.0;
   DATA[1907,3] := 2.0;
   DATA[1907,4] := 262.5609;
   DATA[1907,5] := 8.390669;
   DATA[1907,6] := 332.5814;
   DATA[1907,7] := 2.463461;
   DATA[1907,8] := 2.0;
   DATA[1907,9] := 2.0;
   DATA[1907,10] := 2.0;
   DATA[1907,11] := 19.76759;
   DATA[1907,12] := 2.212215;
   DATA[1907,13] := 793.5466;
   DATA[1907,14] := 1.0;
   DATA[1907,15] := 2.0;
   DATA[1907,16] := 1.0;
   DATA[1907,17] := 1.0;
   DATA[1907,18] := 1.0;
   DATA[1907,19] := 2.0;
   DATA[1907,20] := 148.808;
   DATA[1907,21] := 154.7808;
   DATA[1907,22] := 1.714542;
   DATA[1907,23] := 819.4053;
   DATA[1907,24] := 2.0;
   DATA[1907,25] := 2.0;
   DATA[1907,26] := 7.874135;
   DATA[1907,27] := 143.6042;
   DATA[1907,28] := 262.3045;
   DATA[1907,29] := 12.22763;
   DATA[1907,30] := 1.726737;
   DATA[1907,31] := 1.310491;
   DATA[1907,32] := 0.7352687;
   DATA[1907,33] := 0.3084265;
   DATA[1907,34] := 2.0;
   DATA[1907,35] := 250.3525;
   DATA[1907,36] := 1.730048;
   DATA[1907,37] := 189.1823;
   DATA[1907,38] := 0.000128152;
   DATA[1907,39] := 1.0;
   DATA[1907,40] := 1.0;
   DATA[1908,0] := 2.43026;
   DATA[1908,1] := 859.6354;
   DATA[1908,2] := 2.0;
   DATA[1908,3] := 2.0;
   DATA[1908,4] := 262.5609;
   DATA[1908,5] := 8.390669;
   DATA[1908,6] := 332.5814;
   DATA[1908,7] := 2.463461;
   DATA[1908,8] := 2.0;
   DATA[1908,9] := 2.0;
   DATA[1908,10] := 2.0;
   DATA[1908,11] := 19.76759;
   DATA[1908,12] := 2.21119;
   DATA[1908,13] := 793.5866;
   DATA[1908,14] := 1.0;
   DATA[1908,15] := 2.0;
   DATA[1908,16] := 1.0;
   DATA[1908,17] := 1.0;
   DATA[1908,18] := 1.0;
   DATA[1908,19] := 2.0;
   DATA[1908,20] := 148.808;
   DATA[1908,21] := 154.7808;
   DATA[1908,22] := 1.717361;
   DATA[1908,23] := 819.2899;
   DATA[1908,24] := 2.0;
   DATA[1908,25] := 2.0;
   DATA[1908,26] := 7.874135;
   DATA[1908,27] := 143.8093;
   DATA[1908,28] := 262.3045;
   DATA[1908,29] := 12.22763;
   DATA[1908,30] := 1.728147;
   DATA[1908,31] := 1.29243;
   DATA[1908,32] := 0.7352687;
   DATA[1908,33] := 0.3084265;
   DATA[1908,34] := 2.0;
   DATA[1908,35] := 250.3525;
   DATA[1908,36] := 1.730048;
   DATA[1908,37] := 189.1823;
   DATA[1908,38] := 0.000128152;
   DATA[1908,39] := 1.0;
   DATA[1908,40] := 1.0;
   DATA[1909,0] := 2.436985;
   DATA[1909,1] := 859.1644;
   DATA[1909,2] := 2.0;
   DATA[1909,3] := 2.0;
   DATA[1909,4] := 262.5609;
   DATA[1909,5] := 8.390669;
   DATA[1909,6] := 332.5814;
   DATA[1909,7] := 2.463461;
   DATA[1909,8] := 2.0;
   DATA[1909,9] := 2.0;
   DATA[1909,10] := 2.0;
   DATA[1909,11] := 19.70997;
   DATA[1909,12] := 2.209909;
   DATA[1909,13] := 793.6667;
   DATA[1909,14] := 1.0;
   DATA[1909,15] := 2.0;
   DATA[1909,16] := 1.0;
   DATA[1909,17] := 1.0;
   DATA[1909,18] := 1.0;
   DATA[1909,19] := 2.0;
   DATA[1909,20] := 148.808;
   DATA[1909,21] := 154.7808;
   DATA[1909,22] := 1.717874;
   DATA[1909,23] := 819.4053;
   DATA[1909,24] := 2.0;
   DATA[1909,25] := 2.0;
   DATA[1909,26] := 7.874135;
   DATA[1909,27] := 143.8093;
   DATA[1909,28] := 262.3045;
   DATA[1909,29] := 12.22763;
   DATA[1909,30] := 1.728531;
   DATA[1909,31] := 1.294607;
   DATA[1909,32] := 0.7352687;
   DATA[1909,33] := 0.3084265;
   DATA[1909,34] := 2.0;
   DATA[1909,35] := 250.5768;
   DATA[1909,36] := 1.730048;
   DATA[1909,37] := 189.1823;
   DATA[1909,38] := 0.000128152;
   DATA[1909,39] := 1.0;
   DATA[1909,40] := 1.0;
   DATA[1910,0] := 2.466451;
   DATA[1910,1] := 859.4784;
   DATA[1910,2] := 2.0;
   DATA[1910,3] := 2.0;
   DATA[1910,4] := 262.5609;
   DATA[1910,5] := 8.390669;
   DATA[1910,6] := 332.5814;
   DATA[1910,7] := 2.463461;
   DATA[1910,8] := 2.0;
   DATA[1910,9] := 2.0;
   DATA[1910,10] := 2.0;
   DATA[1910,11] := 19.68436;
   DATA[1910,12] := 2.209909;
   DATA[1910,13] := 793.4664;
   DATA[1910,14] := 1.0;
   DATA[1910,15] := 2.0;
   DATA[1910,16] := 1.0;
   DATA[1910,17] := 1.0;
   DATA[1910,18] := 1.0;
   DATA[1910,19] := 2.0;
   DATA[1910,20] := 148.808;
   DATA[1910,21] := 154.7808;
   DATA[1910,22] := 1.717874;
   DATA[1910,23] := 819.5591;
   DATA[1910,24] := 2.0;
   DATA[1910,25] := 2.0;
   DATA[1910,26] := 7.874135;
   DATA[1910,27] := 143.8093;
   DATA[1910,28] := 262.3045;
   DATA[1910,29] := 12.11228;
   DATA[1910,30] := 1.728531;
   DATA[1910,31] := 1.294607;
   DATA[1910,32] := 0.7352687;
   DATA[1910,33] := 0.3082983;
   DATA[1910,34] := 2.0;
   DATA[1910,35] := 250.5768;
   DATA[1910,36] := 1.730048;
   DATA[1910,37] := 189.4546;
   DATA[1910,38] := 0.000128152;
   DATA[1910,39] := 1.0;
   DATA[1910,40] := 1.0;
   DATA[1911,0] := 2.510009;
   DATA[1911,1] := 859.3214;
   DATA[1911,2] := 2.0;
   DATA[1911,3] := 2.0;
   DATA[1911,4] := 262.5609;
   DATA[1911,5] := 8.390669;
   DATA[1911,6] := 332.5814;
   DATA[1911,7] := 2.465127;
   DATA[1911,8] := 2.0;
   DATA[1911,9] := 2.0;
   DATA[1911,10] := 2.0;
   DATA[1911,11] := 19.65875;
   DATA[1911,12] := 2.209909;
   DATA[1911,13] := 793.7468;
   DATA[1911,14] := 1.0;
   DATA[1911,15] := 2.0;
   DATA[1911,16] := 1.0;
   DATA[1911,17] := 1.0;
   DATA[1911,18] := 1.0;
   DATA[1911,19] := 2.0;
   DATA[1911,20] := 148.808;
   DATA[1911,21] := 154.7808;
   DATA[1911,22] := 1.719027;
   DATA[1911,23] := 819.9436;
   DATA[1911,24] := 2.0;
   DATA[1911,25] := 2.0;
   DATA[1911,26] := 7.874135;
   DATA[1911,27] := 143.8093;
   DATA[1911,28] := 262.3045;
   DATA[1911,29] := 12.11228;
   DATA[1911,30] := 1.728531;
   DATA[1911,31] := 1.289868;
   DATA[1911,32] := 0.7352687;
   DATA[1911,33] := 0.3068251;
   DATA[1911,34] := 2.0;
   DATA[1911,35] := 250.5768;
   DATA[1911,36] := 1.730048;
   DATA[1911,37] := 189.4546;
   DATA[1911,38] := 0.000128152;
   DATA[1911,39] := 1.0;
   DATA[1911,40] := 1.0;
   DATA[1912,0] := 2.551965;
   DATA[1912,1] := 858.9288;
   DATA[1912,2] := 2.0;
   DATA[1912,3] := 2.0;
   DATA[1912,4] := 262.5609;
   DATA[1912,5] := 8.390669;
   DATA[1912,6] := 332.4532;
   DATA[1912,7] := 2.465255;
   DATA[1912,8] := 2.0;
   DATA[1912,9] := 2.0;
   DATA[1912,10] := 2.0;
   DATA[1912,11] := 19.65875;
   DATA[1912,12] := 2.209909;
   DATA[1912,13] := 794.3076;
   DATA[1912,14] := 1.0;
   DATA[1912,15] := 2.0;
   DATA[1912,16] := 1.0;
   DATA[1912,17] := 1.0;
   DATA[1912,18] := 1.0;
   DATA[1912,19] := 2.0;
   DATA[1912,20] := 148.808;
   DATA[1912,21] := 154.7808;
   DATA[1912,22] := 1.719284;
   DATA[1912,23] := 819.636;
   DATA[1912,24] := 2.0;
   DATA[1912,25] := 2.0;
   DATA[1912,26] := 7.874135;
   DATA[1912,27] := 143.8093;
   DATA[1912,28] := 262.3045;
   DATA[1912,29] := 12.11228;
   DATA[1912,30] := 1.728531;
   DATA[1912,31] := 1.289868;
   DATA[1912,32] := 0.7352687;
   DATA[1912,33] := 0.3064407;
   DATA[1912,34] := 2.0;
   DATA[1912,35] := 250.5768;
   DATA[1912,36] := 1.730048;
   DATA[1912,37] := 189.4546;
   DATA[1912,38] := 0.000128152;
   DATA[1912,39] := 1.0;
   DATA[1912,40] := 1.0;
   DATA[1913,0] := 2.590398;
   DATA[1913,1] := 858.9681;
   DATA[1913,2] := 2.0;
   DATA[1913,3] := 2.0;
   DATA[1913,4] := 262.5609;
   DATA[1913,5] := 8.390669;
   DATA[1913,6] := 332.4532;
   DATA[1913,7] := 2.465255;
   DATA[1913,8] := 2.0;
   DATA[1913,9] := 2.0;
   DATA[1913,10] := 2.0;
   DATA[1913,11] := 19.65875;
   DATA[1913,12] := 2.209909;
   DATA[1913,13] := 794.3877;
   DATA[1913,14] := 1.0;
   DATA[1913,15] := 2.0;
   DATA[1913,16] := 1.0;
   DATA[1913,17] := 1.0;
   DATA[1913,18] := 1.0;
   DATA[1913,19] := 2.0;
   DATA[1913,20] := 148.808;
   DATA[1913,21] := 154.7808;
   DATA[1913,22] := 1.720309;
   DATA[1913,23] := 819.8282;
   DATA[1913,24] := 2.0;
   DATA[1913,25] := 2.0;
   DATA[1913,26] := 7.874135;
   DATA[1913,27] := 143.8093;
   DATA[1913,28] := 262.3045;
   DATA[1913,29] := 12.11228;
   DATA[1913,30] := 1.728531;
   DATA[1913,31] := 1.291277;
   DATA[1913,32] := 0.7352687;
   DATA[1913,33] := 0.3065048;
   DATA[1913,34] := 2.0;
   DATA[1913,35] := 250.5768;
   DATA[1913,36] := 1.730048;
   DATA[1913,37] := 189.4546;
   DATA[1913,38] := 0.000128152;
   DATA[1913,39] := 1.0;
   DATA[1913,40] := 1.0;
   DATA[1914,0] := 2.622426;
   DATA[1914,1] := 858.8896;
   DATA[1914,2] := 2.0;
   DATA[1914,3] := 2.0;
   DATA[1914,4] := 262.5609;
   DATA[1914,5] := 8.392271;
   DATA[1914,6] := 332.4532;
   DATA[1914,7] := 2.465255;
   DATA[1914,8] := 2.0;
   DATA[1914,9] := 2.0;
   DATA[1914,10] := 2.0;
   DATA[1914,11] := 19.67155;
   DATA[1914,12] := 2.209653;
   DATA[1914,13] := 794.0673;
   DATA[1914,14] := 1.0;
   DATA[1914,15] := 2.0;
   DATA[1914,16] := 1.0;
   DATA[1914,17] := 1.0;
   DATA[1914,18] := 1.0;
   DATA[1914,19] := 2.0;
   DATA[1914,20] := 148.808;
   DATA[1914,21] := 154.7808;
   DATA[1914,22] := 1.720309;
   DATA[1914,23] := 820.059;
   DATA[1914,24] := 2.0;
   DATA[1914,25] := 2.0;
   DATA[1914,26] := 7.874135;
   DATA[1914,27] := 143.8093;
   DATA[1914,28] := 262.3045;
   DATA[1914,29] := 12.11228;
   DATA[1914,30] := 1.726865;
   DATA[1914,31] := 1.291277;
   DATA[1914,32] := 0.7352687;
   DATA[1914,33] := 0.3086827;
   DATA[1914,34] := 2.0;
   DATA[1914,35] := 250.5768;
   DATA[1914,36] := 1.730048;
   DATA[1914,37] := 189.4546;
   DATA[1914,38] := 0.000128152;
   DATA[1914,39] := 1.0;
   DATA[1914,40] := 1.0;
   DATA[1915,0] := 2.643244;
   DATA[1915,1] := 859.5569;
   DATA[1915,2] := 2.0;
   DATA[1915,3] := 2.0;
   DATA[1915,4] := 262.5609;
   DATA[1915,5] := 8.392271;
   DATA[1915,6] := 332.4532;
   DATA[1915,7] := 2.465255;
   DATA[1915,8] := 2.0;
   DATA[1915,9] := 2.0;
   DATA[1915,10] := 2.0;
   DATA[1915,11] := 19.72277;
   DATA[1915,12] := 2.208884;
   DATA[1915,13] := 794.4678;
   DATA[1915,14] := 1.0;
   DATA[1915,15] := 2.0;
   DATA[1915,16] := 1.0;
   DATA[1915,17] := 1.0;
   DATA[1915,18] := 1.0;
   DATA[1915,19] := 2.0;
   DATA[1915,20] := 148.808;
   DATA[1915,21] := 154.7808;
   DATA[1915,22] := 1.720309;
   DATA[1915,23] := 820.5204;
   DATA[1915,24] := 2.0;
   DATA[1915,25] := 2.0;
   DATA[1915,26] := 7.874135;
   DATA[1915,27] := 143.8093;
   DATA[1915,28] := 262.3045;
   DATA[1915,29] := 12.11228;
   DATA[1915,30] := 1.724942;
   DATA[1915,31] := 1.291533;
   DATA[1915,32] := 0.7352687;
   DATA[1915,33] := 0.3086827;
   DATA[1915,34] := 2.0;
   DATA[1915,35] := 250.5768;
   DATA[1915,36] := 1.730048;
   DATA[1915,37] := 189.1823;
   DATA[1915,38] := 0.000128152;
   DATA[1915,39] := 1.0;
   DATA[1915,40] := 1.0;
   DATA[1916,0] := 2.657656;
   DATA[1916,1] := 859.6747;
   DATA[1916,2] := 2.0;
   DATA[1916,3] := 2.0;
   DATA[1916,4] := 262.5609;
   DATA[1916,5] := 8.392271;
   DATA[1916,6] := 332.4532;
   DATA[1916,7] := 2.465255;
   DATA[1916,8] := 2.0;
   DATA[1916,9] := 2.0;
   DATA[1916,10] := 2.0;
   DATA[1916,11] := 19.72277;
   DATA[1916,12] := 2.208884;
   DATA[1916,13] := 794.3076;
   DATA[1916,14] := 1.0;
   DATA[1916,15] := 2.0;
   DATA[1916,16] := 1.0;
   DATA[1916,17] := 1.0;
   DATA[1916,18] := 1.0;
   DATA[1916,19] := 2.0;
   DATA[1916,20] := 148.808;
   DATA[1916,21] := 154.7808;
   DATA[1916,22] := 1.720309;
   DATA[1916,23] := 820.7126;
   DATA[1916,24] := 2.0;
   DATA[1916,25] := 2.0;
   DATA[1916,26] := 7.874135;
   DATA[1916,27] := 143.8093;
   DATA[1916,28] := 262.1764;
   DATA[1916,29] := 12.11228;
   DATA[1916,30] := 1.724942;
   DATA[1916,31] := 1.291533;
   DATA[1916,32] := 0.7352687;
   DATA[1916,33] := 0.3070813;
   DATA[1916,34] := 2.0;
   DATA[1916,35] := 250.5768;
   DATA[1916,36] := 1.730048;
   DATA[1916,37] := 189.1823;
   DATA[1916,38] := 0.000128152;
   DATA[1916,39] := 1.0;
   DATA[1916,40] := 1.0;
   DATA[1917,0] := 2.660539;
   DATA[1917,1] := 859.7532;
   DATA[1917,2] := 2.0;
   DATA[1917,3] := 2.0;
   DATA[1917,4] := 262.5609;
   DATA[1917,5] := 8.392271;
   DATA[1917,6] := 332.4532;
   DATA[1917,7] := 2.462564;
   DATA[1917,8] := 2.0;
   DATA[1917,9] := 2.0;
   DATA[1917,10] := 2.0;
   DATA[1917,11] := 19.72277;
   DATA[1917,12] := 2.208884;
   DATA[1917,13] := 794.1473;
   DATA[1917,14] := 1.0;
   DATA[1917,15] := 2.0;
   DATA[1917,16] := 1.0;
   DATA[1917,17] := 1.0;
   DATA[1917,18] := 1.0;
   DATA[1917,19] := 2.0;
   DATA[1917,20] := 148.808;
   DATA[1917,21] := 154.7808;
   DATA[1917,22] := 1.717233;
   DATA[1917,23] := 821.4817;
   DATA[1917,24] := 2.0;
   DATA[1917,25] := 2.0;
   DATA[1917,26] := 7.874135;
   DATA[1917,27] := 143.8093;
   DATA[1917,28] := 262.1764;
   DATA[1917,29] := 12.11228;
   DATA[1917,30] := 1.724942;
   DATA[1917,31] := 1.291533;
   DATA[1917,32] := 0.7352687;
   DATA[1917,33] := 0.3079781;
   DATA[1917,34] := 2.0;
   DATA[1917,35] := 250.4646;
   DATA[1917,36] := 1.730048;
   DATA[1917,37] := 189.1823;
   DATA[1917,38] := 0.000128152;
   DATA[1917,39] := 1.0;
   DATA[1917,40] := 1.0;
   DATA[1918,0] := 2.634917;
   DATA[1918,1] := 859.2429;
   DATA[1918,2] := 2.0;
   DATA[1918,3] := 2.0;
   DATA[1918,4] := 262.5609;
   DATA[1918,5] := 8.395155;
   DATA[1918,6] := 332.4532;
   DATA[1918,7] := 2.462564;
   DATA[1918,8] := 2.0;
   DATA[1918,9] := 2.0;
   DATA[1918,10] := 2.0;
   DATA[1918,11] := 19.75479;
   DATA[1918,12] := 2.208884;
   DATA[1918,13] := 794.2675;
   DATA[1918,14] := 1.0;
   DATA[1918,15] := 2.0;
   DATA[1918,16] := 1.0;
   DATA[1918,17] := 1.0;
   DATA[1918,18] := 1.0;
   DATA[1918,19] := 2.0;
   DATA[1918,20] := 148.808;
   DATA[1918,21] := 154.7808;
   DATA[1918,22] := 1.717233;
   DATA[1918,23] := 821.7124;
   DATA[1918,24] := 2.0;
   DATA[1918,25] := 2.0;
   DATA[1918,26] := 7.874135;
   DATA[1918,27] := 143.8093;
   DATA[1918,28] := 262.1764;
   DATA[1918,29] := 12.11228;
   DATA[1918,30] := 1.724942;
   DATA[1918,31] := 1.3005;
   DATA[1918,32] := 0.7352687;
   DATA[1918,33] := 0.3084905;
   DATA[1918,34] := 2.0;
   DATA[1918,35] := 250.4166;
   DATA[1918,36] := 1.730048;
   DATA[1918,37] := 189.1823;
   DATA[1918,38] := 0.000128152;
   DATA[1918,39] := 1.0;
   DATA[1918,40] := 1.0;
   DATA[1919,0] := 2.623387;
   DATA[1919,1] := 859.4391;
   DATA[1919,2] := 2.0;
   DATA[1919,3] := 2.0;
   DATA[1919,4] := 262.5609;
   DATA[1919,5] := 8.395155;
   DATA[1919,6] := 332.4532;
   DATA[1919,7] := 2.462564;
   DATA[1919,8] := 2.0;
   DATA[1919,9] := 2.0;
   DATA[1919,10] := 2.0;
   DATA[1919,11] := 19.7804;
   DATA[1919,12] := 2.208884;
   DATA[1919,13] := 794.2675;
   DATA[1919,14] := 1.0;
   DATA[1919,15] := 2.0;
   DATA[1919,16] := 1.0;
   DATA[1919,17] := 1.0;
   DATA[1919,18] := 1.0;
   DATA[1919,19] := 2.0;
   DATA[1919,20] := 148.808;
   DATA[1919,21] := 154.7808;
   DATA[1919,22] := 1.717233;
   DATA[1919,23] := 821.8662;
   DATA[1919,24] := 2.0;
   DATA[1919,25] := 2.0;
   DATA[1919,26] := 7.874135;
   DATA[1919,27] := 143.8093;
   DATA[1919,28] := 262.1764;
   DATA[1919,29] := 12.11228;
   DATA[1919,30] := 1.724942;
   DATA[1919,31] := 1.298194;
   DATA[1919,32] := 0.7352687;
   DATA[1919,33] := 0.3084905;
   DATA[1919,34] := 2.0;
   DATA[1919,35] := 250.3845;
   DATA[1919,36] := 1.730048;
   DATA[1919,37] := 189.1823;
   DATA[1919,38] := 0.000128152;
   DATA[1919,39] := 1.0;
   DATA[1919,40] := 1.0;
   DATA[1920,0] := 2.61634;
   DATA[1920,1] := 859.3214;
   DATA[1920,2] := 2.0;
   DATA[1920,3] := 2.0;
   DATA[1920,4] := 262.5609;
   DATA[1920,5] := 8.395155;
   DATA[1920,6] := 332.4532;
   DATA[1920,7] := 2.462564;
   DATA[1920,8] := 2.0;
   DATA[1920,9] := 2.0;
   DATA[1920,10] := 2.0;
   DATA[1920,11] := 19.7804;
   DATA[1920,12] := 2.208884;
   DATA[1920,13] := 794.1073;
   DATA[1920,14] := 1.0;
   DATA[1920,15] := 2.0;
   DATA[1920,16] := 1.0;
   DATA[1920,17] := 1.0;
   DATA[1920,18] := 1.0;
   DATA[1920,19] := 2.0;
   DATA[1920,20] := 148.808;
   DATA[1920,21] := 154.7808;
   DATA[1920,22] := 1.717233;
   DATA[1920,23] := 822.3661;
   DATA[1920,24] := 2.0;
   DATA[1920,25] := 2.0;
   DATA[1920,26] := 7.874135;
   DATA[1920,27] := 143.8093;
   DATA[1920,28] := 262.1764;
   DATA[1920,29] := 12.11228;
   DATA[1920,30] := 1.724942;
   DATA[1920,31] := 1.283207;
   DATA[1920,32] := 0.7352687;
   DATA[1920,33] := 0.3084905;
   DATA[1920,34] := 2.0;
   DATA[1920,35] := 250.3845;
   DATA[1920,36] := 1.730048;
   DATA[1920,37] := 189.1823;
   DATA[1920,38] := 0.000128152;
   DATA[1920,39] := 1.0;
   DATA[1920,40] := 1.0;
   DATA[1921,0] := 2.614419;
   DATA[1921,1] := 859.7139;
   DATA[1921,2] := 2.0;
   DATA[1921,3] := 2.0;
   DATA[1921,4] := 262.5609;
   DATA[1921,5] := 8.395155;
   DATA[1921,6] := 332.4532;
   DATA[1921,7] := 2.462564;
   DATA[1921,8] := 2.0;
   DATA[1921,9] := 2.0;
   DATA[1921,10] := 2.0;
   DATA[1921,11] := 19.7804;
   DATA[1921,12] := 2.208884;
   DATA[1921,13] := 793.9871;
   DATA[1921,14] := 1.0;
   DATA[1921,15] := 2.0;
   DATA[1921,16] := 1.0;
   DATA[1921,17] := 1.0;
   DATA[1921,18] := 1.0;
   DATA[1921,19] := 2.0;
   DATA[1921,20] := 148.808;
   DATA[1921,21] := 154.6783;
   DATA[1921,22] := 1.717233;
   DATA[1921,23] := 822.7121;
   DATA[1921,24] := 2.0;
   DATA[1921,25] := 2.0;
   DATA[1921,26] := 7.874135;
   DATA[1921,27] := 143.8093;
   DATA[1921,28] := 262.1764;
   DATA[1921,29] := 12.11228;
   DATA[1921,30] := 1.724942;
   DATA[1921,31] := 1.281798;
   DATA[1921,32] := 0.7352687;
   DATA[1921,33] := 0.3084905;
   DATA[1921,34] := 2.0;
   DATA[1921,35] := 250.3845;
   DATA[1921,36] := 1.730048;
   DATA[1921,37] := 189.1823;
   DATA[1921,38] := 0.000128152;
   DATA[1921,39] := 1.0;
   DATA[1921,40] := 1.0;
   DATA[1922,0] := 2.601608;
   DATA[1922,1] := 859.5176;
   DATA[1922,2] := 2.0;
   DATA[1922,3] := 2.0;
   DATA[1922,4] := 262.5609;
   DATA[1922,5] := 8.395155;
   DATA[1922,6] := 332.4019;
   DATA[1922,7] := 2.462564;
   DATA[1922,8] := 2.0;
   DATA[1922,9] := 2.0;
   DATA[1922,10] := 2.0;
   DATA[1922,11] := 19.7804;
   DATA[1922,12] := 2.208884;
   DATA[1922,13] := 794.1874;
   DATA[1922,14] := 1.0;
   DATA[1922,15] := 2.0;
   DATA[1922,16] := 1.0;
   DATA[1922,17] := 1.0;
   DATA[1922,18] := 1.0;
   DATA[1922,19] := 2.0;
   DATA[1922,20] := 148.808;
   DATA[1922,21] := 154.5501;
   DATA[1922,22] := 1.717233;
   DATA[1922,23] := 823.0582;
   DATA[1922,24] := 2.0;
   DATA[1922,25] := 2.0;
   DATA[1922,26] := 7.874135;
   DATA[1922,27] := 143.8093;
   DATA[1922,28] := 262.1764;
   DATA[1922,29] := 12.11228;
   DATA[1922,30] := 1.724942;
   DATA[1922,31] := 1.287947;
   DATA[1922,32] := 0.7352687;
   DATA[1922,33] := 0.3084905;
   DATA[1922,34] := 2.0;
   DATA[1922,35] := 250.3845;
   DATA[1922,36] := 1.730048;
   DATA[1922,37] := 189.1022;
   DATA[1922,38] := 0.000128152;
   DATA[1922,39] := 1.0;
   DATA[1922,40] := 1.0;
   DATA[1923,0] := 2.582391;
   DATA[1923,1] := 859.8317;
   DATA[1923,2] := 2.0;
   DATA[1923,3] := 2.0;
   DATA[1923,4] := 262.5609;
   DATA[1923,5] := 8.395155;
   DATA[1923,6] := 332.3507;
   DATA[1923,7] := 2.465383;
   DATA[1923,8] := 2.0;
   DATA[1923,9] := 2.0;
   DATA[1923,10] := 2.0;
   DATA[1923,11] := 19.7804;
   DATA[1923,12] := 2.208884;
   DATA[1923,13] := 794.3877;
   DATA[1923,14] := 1.0;
   DATA[1923,15] := 2.0;
   DATA[1923,16] := 1.0;
   DATA[1923,17] := 1.0;
   DATA[1923,18] := 1.0;
   DATA[1923,19] := 2.0;
   DATA[1923,20] := 148.808;
   DATA[1923,21] := 154.5501;
   DATA[1923,22] := 1.717233;
   DATA[1923,23] := 822.8659;
   DATA[1923,24] := 2.0;
   DATA[1923,25] := 2.0;
   DATA[1923,26] := 7.874135;
   DATA[1923,27] := 143.8093;
   DATA[1923,28] := 262.1764;
   DATA[1923,29] := 12.11228;
   DATA[1923,30] := 1.724942;
   DATA[1923,31] := 1.307288;
   DATA[1923,32] := 0.7352687;
   DATA[1923,33] := 0.3084905;
   DATA[1923,34] := 2.0;
   DATA[1923,35] := 250.3845;
   DATA[1923,36] := 1.730048;
   DATA[1923,37] := 188.974;
   DATA[1923,38] := 0.000128152;
   DATA[1923,39] := 1.0;
   DATA[1923,40] := 1.0;
   DATA[1924,0] := 2.566377;
   DATA[1924,1] := 859.7139;
   DATA[1924,2] := 2.0;
   DATA[1924,3] := 2.0;
   DATA[1924,4] := 262.5609;
   DATA[1924,5] := 8.395155;
   DATA[1924,6] := 332.3507;
   DATA[1924,7] := 2.465383;
   DATA[1924,8] := 2.0;
   DATA[1924,9] := 2.0;
   DATA[1924,10] := 2.0;
   DATA[1924,11] := 19.77079;
   DATA[1924,12] := 2.208884;
   DATA[1924,13] := 794.3076;
   DATA[1924,14] := 1.0;
   DATA[1924,15] := 2.0;
   DATA[1924,16] := 1.0;
   DATA[1924,17] := 1.0;
   DATA[1924,18] := 1.0;
   DATA[1924,19] := 2.0;
   DATA[1924,20] := 148.808;
   DATA[1924,21] := 154.5501;
   DATA[1924,22] := 1.717233;
   DATA[1924,23] := 823.2889;
   DATA[1924,24] := 2.0;
   DATA[1924,25] := 2.0;
   DATA[1924,26] := 7.874135;
   DATA[1924,27] := 143.8093;
   DATA[1924,28] := 262.2404;
   DATA[1924,29] := 12.11228;
   DATA[1924,30] := 1.724942;
   DATA[1924,31] := 1.307288;
   DATA[1924,32] := 0.7352687;
   DATA[1924,33] := 0.3084905;
   DATA[1924,34] := 2.0;
   DATA[1924,35] := 250.3845;
   DATA[1924,36] := 1.730048;
   DATA[1924,37] := 188.974;
   DATA[1924,38] := 0.000128152;
   DATA[1924,39] := 1.0;
   DATA[1924,40] := 1.0;
   DATA[1925,0] := 2.549082;
   DATA[1925,1] := 859.7532;
   DATA[1925,2] := 2.0;
   DATA[1925,3] := 2.0;
   DATA[1925,4] := 262.5609;
   DATA[1925,5] := 8.395155;
   DATA[1925,6] := 332.3507;
   DATA[1925,7] := 2.465383;
   DATA[1925,8] := 2.0;
   DATA[1925,9] := 2.0;
   DATA[1925,10] := 2.0;
   DATA[1925,11] := 19.73878;
   DATA[1925,12] := 2.208884;
   DATA[1925,13] := 794.2675;
   DATA[1925,14] := 1.0;
   DATA[1925,15] := 2.0;
   DATA[1925,16] := 1.0;
   DATA[1925,17] := 1.0;
   DATA[1925,18] := 1.0;
   DATA[1925,19] := 2.0;
   DATA[1925,20] := 148.808;
   DATA[1925,21] := 154.5501;
   DATA[1925,22] := 1.717233;
   DATA[1925,23] := 823.4042;
   DATA[1925,24] := 2.0;
   DATA[1925,25] := 2.0;
   DATA[1925,26] := 7.874135;
   DATA[1925,27] := 143.8093;
   DATA[1925,28] := 262.2404;
   DATA[1925,29] := 12.11228;
   DATA[1925,30] := 1.72302;
   DATA[1925,31] := 1.302293;
   DATA[1925,32] := 0.7352687;
   DATA[1925,33] := 0.3084905;
   DATA[1925,34] := 2.0;
   DATA[1925,35] := 250.2563;
   DATA[1925,36] := 1.730048;
   DATA[1925,37] := 188.974;
   DATA[1925,38] := 0.000128152;
   DATA[1925,39] := 1.0;
   DATA[1925,40] := 1.0;
   DATA[1926,0] := 2.533068;
   DATA[1926,1] := 859.6354;
   DATA[1926,2] := 2.0;
   DATA[1926,3] := 2.0;
   DATA[1926,4] := 262.5609;
   DATA[1926,5] := 8.395155;
   DATA[1926,6] := 332.3507;
   DATA[1926,7] := 2.465383;
   DATA[1926,8] := 2.0;
   DATA[1926,9] := 2.0;
   DATA[1926,10] := 2.0;
   DATA[1926,11] := 19.73878;
   DATA[1926,12] := 2.208884;
   DATA[1926,13] := 793.9471;
   DATA[1926,14] := 1.0;
   DATA[1926,15] := 2.0;
   DATA[1926,16] := 1.0;
   DATA[1926,17] := 1.0;
   DATA[1926,18] := 1.0;
   DATA[1926,19] := 2.0;
   DATA[1926,20] := 148.808;
   DATA[1926,21] := 154.5501;
   DATA[1926,22] := 1.717233;
   DATA[1926,23] := 823.2889;
   DATA[1926,24] := 2.0;
   DATA[1926,25] := 2.0;
   DATA[1926,26] := 7.874135;
   DATA[1926,27] := 143.8093;
   DATA[1926,28] := 262.2404;
   DATA[1926,29] := 12.11228;
   DATA[1926,30] := 1.72302;
   DATA[1926,31] := 1.282311;
   DATA[1926,32] := 0.7352687;
   DATA[1926,33] := 0.3083624;
   DATA[1926,34] := 2.0;
   DATA[1926,35] := 250.2563;
   DATA[1926,36] := 1.730048;
   DATA[1926,37] := 188.974;
   DATA[1926,38] := 0.000128152;
   DATA[1926,39] := 1.0;
   DATA[1926,40] := 1.0;
   DATA[1927,0] := 2.520257;
   DATA[1927,1] := 859.7532;
   DATA[1927,2] := 2.0;
   DATA[1927,3] := 2.0;
   DATA[1927,4] := 262.4648;
   DATA[1927,5] := 8.395155;
   DATA[1927,6] := 332.3507;
   DATA[1927,7] := 2.465767;
   DATA[1927,8] := 2.0;
   DATA[1927,9] := 2.0;
   DATA[1927,10] := 2.0;
   DATA[1927,11] := 19.73878;
   DATA[1927,12] := 2.208884;
   DATA[1927,13] := 794.3076;
   DATA[1927,14] := 1.0;
   DATA[1927,15] := 2.0;
   DATA[1927,16] := 1.0;
   DATA[1927,17] := 1.0;
   DATA[1927,18] := 1.0;
   DATA[1927,19] := 2.0;
   DATA[1927,20] := 148.808;
   DATA[1927,21] := 154.5501;
   DATA[1927,22] := 1.717233;
   DATA[1927,23] := 823.5965;
   DATA[1927,24] := 2.0;
   DATA[1927,25] := 2.0;
   DATA[1927,26] := 7.874135;
   DATA[1927,27] := 143.8093;
   DATA[1927,28] := 262.2404;
   DATA[1927,29] := 12.11228;
   DATA[1927,30] := 1.72302;
   DATA[1927,31] := 1.271935;
   DATA[1927,32] := 0.7352687;
   DATA[1927,33] := 0.3083624;
   DATA[1927,34] := 2.0;
   DATA[1927,35] := 250.2563;
   DATA[1927,36] := 1.730048;
   DATA[1927,37] := 188.974;
   DATA[1927,38] := 0.000128152;
   DATA[1927,39] := 1.0;
   DATA[1927,40] := 1.0;
   DATA[1928,0] := 2.505525;
   DATA[1928,1] := 859.6354;
   DATA[1928,2] := 2.0;
   DATA[1928,3] := 2.0;
   DATA[1928,4] := 262.4648;
   DATA[1928,5] := 8.395155;
   DATA[1928,6] := 332.3507;
   DATA[1928,7] := 2.466024;
   DATA[1928,8] := 2.0;
   DATA[1928,9] := 2.0;
   DATA[1928,10] := 2.0;
   DATA[1928,11] := 19.73878;
   DATA[1928,12] := 2.208884;
   DATA[1928,13] := 794.1874;
   DATA[1928,14] := 1.0;
   DATA[1928,15] := 2.0;
   DATA[1928,16] := 1.0;
   DATA[1928,17] := 1.0;
   DATA[1928,18] := 1.0;
   DATA[1928,19] := 2.0;
   DATA[1928,20] := 148.808;
   DATA[1928,21] := 154.5501;
   DATA[1928,22] := 1.717233;
   DATA[1928,23] := 823.6734;
   DATA[1928,24] := 2.0;
   DATA[1928,25] := 2.0;
   DATA[1928,26] := 7.874135;
   DATA[1928,27] := 143.8093;
   DATA[1928,28] := 262.2404;
   DATA[1928,29] := 12.11228;
   DATA[1928,30] := 1.72302;
   DATA[1928,31] := 1.271551;
   DATA[1928,32] := 0.7352687;
   DATA[1928,33] := 0.3083624;
   DATA[1928,34] := 2.0;
   DATA[1928,35] := 250.1762;
   DATA[1928,36] := 1.730048;
   DATA[1928,37] := 188.974;
   DATA[1928,38] := 0.000128152;
   DATA[1928,39] := 1.0;
   DATA[1928,40] := 1.0;
   DATA[1929,0] := 2.491112;
   DATA[1929,1] := 859.7532;
   DATA[1929,2] := 2.0;
   DATA[1929,3] := 2.0;
   DATA[1929,4] := 262.4648;
   DATA[1929,5] := 8.395155;
   DATA[1929,6] := 332.3507;
   DATA[1929,7] := 2.466024;
   DATA[1929,8] := 2.0;
   DATA[1929,9] := 2.0;
   DATA[1929,10] := 2.0;
   DATA[1929,11] := 19.73878;
   DATA[1929,12] := 2.209653;
   DATA[1929,13] := 793.7869;
   DATA[1929,14] := 1.0;
   DATA[1929,15] := 2.0;
   DATA[1929,16] := 1.0;
   DATA[1929,17] := 1.0;
   DATA[1929,18] := 1.0;
   DATA[1929,19] := 2.0;
   DATA[1929,20] := 148.808;
   DATA[1929,21] := 154.5501;
   DATA[1929,22] := 1.719156;
   DATA[1929,23] := 823.7119;
   DATA[1929,24] := 2.0;
   DATA[1929,25] := 2.0;
   DATA[1929,26] := 7.874135;
   DATA[1929,27] := 143.8093;
   DATA[1929,28] := 262.2404;
   DATA[1929,29] := 12.11228;
   DATA[1929,30] := 1.72302;
   DATA[1929,31] := 1.262713;
   DATA[1929,32] := 0.7352687;
   DATA[1929,33] := 0.3083624;
   DATA[1929,34] := 2.0;
   DATA[1929,35] := 250.1762;
   DATA[1929,36] := 1.730048;
   DATA[1929,37] := 188.974;
   DATA[1929,38] := 0.000128152;
   DATA[1929,39] := 1.0;
   DATA[1929,40] := 1.0;
   DATA[1930,0] := 2.471896;
   DATA[1930,1] := 859.7139;
   DATA[1930,2] := 2.0;
   DATA[1930,3] := 2.0;
   DATA[1930,4] := 262.4648;
   DATA[1930,5] := 8.395155;
   DATA[1930,6] := 332.3507;
   DATA[1930,7] := 2.466024;
   DATA[1930,8] := 2.0;
   DATA[1930,9] := 2.0;
   DATA[1930,10] := 2.0;
   DATA[1930,11] := 19.73878;
   DATA[1930,12] := 2.209653;
   DATA[1930,13] := 793.867;
   DATA[1930,14] := 1.0;
   DATA[1930,15] := 2.0;
   DATA[1930,16] := 1.0;
   DATA[1930,17] := 1.0;
   DATA[1930,18] := 1.0;
   DATA[1930,19] := 2.0;
   DATA[1930,20] := 148.808;
   DATA[1930,21] := 154.5501;
   DATA[1930,22] := 1.719156;
   DATA[1930,23] := 824.2502;
   DATA[1930,24] := 2.0;
   DATA[1930,25] := 2.0;
   DATA[1930,26] := 7.874135;
   DATA[1930,27] := 143.8093;
   DATA[1930,28] := 262.2404;
   DATA[1930,29] := 12.11228;
   DATA[1930,30] := 1.724045;
   DATA[1930,31] := 1.265659;
   DATA[1930,32] := 0.7352687;
   DATA[1930,33] := 0.3083624;
   DATA[1930,34] := 2.0;
   DATA[1930,35] := 250.1762;
   DATA[1930,36] := 1.730048;
   DATA[1930,37] := 189.1022;
   DATA[1930,38] := 0.000128152;
   DATA[1930,39] := 1.0;
   DATA[1930,40] := 1.0;
   DATA[1931,0] := 2.459085;
   DATA[1931,1] := 860.0672;
   DATA[1931,2] := 2.0;
   DATA[1931,3] := 2.0;
   DATA[1931,4] := 262.4648;
   DATA[1931,5] := 8.395155;
   DATA[1931,6] := 332.325;
   DATA[1931,7] := 2.465255;
   DATA[1931,8] := 2.0;
   DATA[1931,9] := 2.0;
   DATA[1931,10] := 2.0;
   DATA[1931,11] := 19.73878;
   DATA[1931,12] := 2.209653;
   DATA[1931,13] := 794.1874;
   DATA[1931,14] := 1.0;
   DATA[1931,15] := 2.0;
   DATA[1931,16] := 1.0;
   DATA[1931,17] := 1.0;
   DATA[1931,18] := 1.0;
   DATA[1931,19] := 2.0;
   DATA[1931,20] := 148.808;
   DATA[1931,21] := 154.5501;
   DATA[1931,22] := 1.719156;
   DATA[1931,23] := 824.0195;
   DATA[1931,24] := 2.0;
   DATA[1931,25] := 2.0;
   DATA[1931,26] := 7.874135;
   DATA[1931,27] := 143.8093;
   DATA[1931,28] := 262.2404;
   DATA[1931,29] := 12.11228;
   DATA[1931,30] := 1.724686;
   DATA[1931,31] := 1.26694;
   DATA[1931,32] := 0.7352687;
   DATA[1931,33] := 0.3083624;
   DATA[1931,34] := 2.0;
   DATA[1931,35] := 250.1762;
   DATA[1931,36] := 1.730048;
   DATA[1931,37] := 189.1022;
   DATA[1931,38] := 0.000128152;
   DATA[1931,39] := 1.0;
   DATA[1931,40] := 1.0;
   DATA[1932,0] := 2.44275;
   DATA[1932,1] := 860.2242;
   DATA[1932,2] := 2.0;
   DATA[1932,3] := 2.0;
   DATA[1932,4] := 262.4648;
   DATA[1932,5] := 8.395155;
   DATA[1932,6] := 332.1969;
   DATA[1932,7] := 2.465255;
   DATA[1932,8] := 2.0;
   DATA[1932,9] := 2.0;
   DATA[1932,10] := 2.0;
   DATA[1932,11] := 19.69076;
   DATA[1932,12] := 2.208884;
   DATA[1932,13] := 793.907;
   DATA[1932,14] := 1.0;
   DATA[1932,15] := 2.0;
   DATA[1932,16] := 1.0;
   DATA[1932,17] := 1.0;
   DATA[1932,18] := 1.0;
   DATA[1932,19] := 2.0;
   DATA[1932,20] := 148.808;
   DATA[1932,21] := 154.5501;
   DATA[1932,22] := 1.719156;
   DATA[1932,23] := 824.2117;
   DATA[1932,24] := 2.0;
   DATA[1932,25] := 2.0;
   DATA[1932,26] := 7.874135;
   DATA[1932,27] := 143.8093;
   DATA[1932,28] := 262.2404;
   DATA[1932,29] := 12.11228;
   DATA[1932,30] := 1.724814;
   DATA[1932,31] := 1.270911;
   DATA[1932,32] := 0.7352687;
   DATA[1932,33] := 0.3083624;
   DATA[1932,34] := 2.0;
   DATA[1932,35] := 250.1762;
   DATA[1932,36] := 1.730048;
   DATA[1932,37] := 189.1022;
   DATA[1932,38] := 0.000128152;
   DATA[1932,39] := 1.0;
   DATA[1932,40] := 1.0;
   DATA[1933,0] := 2.433462;
   DATA[1933,1] := 860.4597;
   DATA[1933,2] := 2.0;
   DATA[1933,3] := 2.0;
   DATA[1933,4] := 262.4648;
   DATA[1933,5] := 8.393553;
   DATA[1933,6] := 332.1969;
   DATA[1933,7] := 2.465255;
   DATA[1933,8] := 2.0;
   DATA[1933,9] := 2.0;
   DATA[1933,10] := 2.0;
   DATA[1933,11] := 19.69076;
   DATA[1933,12] := 2.208884;
   DATA[1933,13] := 794.3076;
   DATA[1933,14] := 1.0;
   DATA[1933,15] := 2.0;
   DATA[1933,16] := 1.0;
   DATA[1933,17] := 1.0;
   DATA[1933,18] := 1.0;
   DATA[1933,19] := 2.0;
   DATA[1933,20] := 148.808;
   DATA[1933,21] := 154.5501;
   DATA[1933,22] := 1.718643;
   DATA[1933,23] := 824.0964;
   DATA[1933,24] := 2.0;
   DATA[1933,25] := 2.0;
   DATA[1933,26] := 7.874135;
   DATA[1933,27] := 143.8093;
   DATA[1933,28] := 262.2404;
   DATA[1933,29] := 12.11228;
   DATA[1933,30] := 1.724814;
   DATA[1933,31] := 1.281158;
   DATA[1933,32] := 0.7352687;
   DATA[1933,33] := 0.3083624;
   DATA[1933,34] := 2.0;
   DATA[1933,35] := 250.1762;
   DATA[1933,36] := 1.730048;
   DATA[1933,37] := 189.1022;
   DATA[1933,38] := 0.000128152;
   DATA[1933,39] := 1.0;
   DATA[1933,40] := 1.0;
   DATA[1934,0] := 2.425135;
   DATA[1934,1] := 860.6167;
   DATA[1934,2] := 2.0;
   DATA[1934,3] := 2.0;
   DATA[1934,4] := 262.4648;
   DATA[1934,5] := 8.391951;
   DATA[1934,6] := 332.1969;
   DATA[1934,7] := 2.465255;
   DATA[1934,8] := 2.0;
   DATA[1934,9] := 2.0;
   DATA[1934,10] := 2.0;
   DATA[1934,11] := 19.69076;
   DATA[1934,12] := 2.208884;
   DATA[1934,13] := 794.5479;
   DATA[1934,14] := 1.0;
   DATA[1934,15] := 2.0;
   DATA[1934,16] := 1.0;
   DATA[1934,17] := 1.0;
   DATA[1934,18] := 1.0;
   DATA[1934,19] := 2.0;
   DATA[1934,20] := 148.808;
   DATA[1934,21] := 154.5501;
   DATA[1934,22] := 1.71608;
   DATA[1934,23] := 824.4809;
   DATA[1934,24] := 2.0;
   DATA[1934,25] := 2.0;
   DATA[1934,26] := 7.874135;
   DATA[1934,27] := 143.9375;
   DATA[1934,28] := 262.2404;
   DATA[1934,29] := 12.11228;
   DATA[1934,30] := 1.724814;
   DATA[1934,31] := 1.292174;
   DATA[1934,32] := 0.7352687;
   DATA[1934,33] := 0.3083624;
   DATA[1934,34] := 2.0;
   DATA[1934,35] := 250.1762;
   DATA[1934,36] := 1.730048;
   DATA[1934,37] := 189.1022;
   DATA[1934,38] := 0.000128152;
   DATA[1934,39] := 1.0;
   DATA[1934,40] := 1.0;
   DATA[1935,0] := 2.425135;
   DATA[1935,1] := 860.6167;
   DATA[1935,2] := 2.0;
   DATA[1935,3] := 2.0;
   DATA[1935,4] := 262.4648;
   DATA[1935,5] := 8.391951;
   DATA[1935,6] := 332.1969;
   DATA[1935,7] := 2.465255;
   DATA[1935,8] := 2.0;
   DATA[1935,9] := 2.0;
   DATA[1935,10] := 2.0;
   DATA[1935,11] := 19.72277;
   DATA[1935,12] := 2.208884;
   DATA[1935,13] := 794.3877;
   DATA[1935,14] := 1.0;
   DATA[1935,15] := 2.0;
   DATA[1935,16] := 1.0;
   DATA[1935,17] := 1.0;
   DATA[1935,18] := 1.0;
   DATA[1935,19] := 2.0;
   DATA[1935,20] := 148.808;
   DATA[1935,21] := 154.5501;
   DATA[1935,22] := 1.715824;
   DATA[1935,23] := 824.5963;
   DATA[1935,24] := 2.0;
   DATA[1935,25] := 2.0;
   DATA[1935,26] := 7.874135;
   DATA[1935,27] := 143.9375;
   DATA[1935,28] := 262.2404;
   DATA[1935,29] := 12.11228;
   DATA[1935,30] := 1.723789;
   DATA[1935,31] := 1.29243;
   DATA[1935,32] := 0.7352687;
   DATA[1935,33] := 0.3083624;
   DATA[1935,34] := 2.0;
   DATA[1935,35] := 250.1762;
   DATA[1935,36] := 1.730048;
   DATA[1935,37] := 189.1022;
   DATA[1935,38] := 0.000128152;
   DATA[1935,39] := 1.0;
   DATA[1935,40] := 1.0;
   DATA[1936,0] := 2.444031;
   DATA[1936,1] := 860.3027;
   DATA[1936,2] := 2.0;
   DATA[1936,3] := 2.0;
   DATA[1936,4] := 262.4648;
   DATA[1936,5] := 8.391951;
   DATA[1936,6] := 332.1969;
   DATA[1936,7] := 2.463461;
   DATA[1936,8] := 2.0;
   DATA[1936,9] := 2.0;
   DATA[1936,10] := 2.0;
   DATA[1936,11] := 19.73238;
   DATA[1936,12] := 2.208884;
   DATA[1936,13] := 795.1086;
   DATA[1936,14] := 1.0;
   DATA[1936,15] := 2.0;
   DATA[1936,16] := 1.0;
   DATA[1936,17] := 1.0;
   DATA[1936,18] := 1.0;
   DATA[1936,19] := 2.0;
   DATA[1936,20] := 148.808;
   DATA[1936,21] := 154.7552;
   DATA[1936,22] := 1.715824;
   DATA[1936,23] := 824.9808;
   DATA[1936,24] := 2.0;
   DATA[1936,25] := 2.0;
   DATA[1936,26] := 7.874135;
   DATA[1936,27] := 143.9375;
   DATA[1936,28] := 262.2404;
   DATA[1936,29] := 12.11228;
   DATA[1936,30] := 1.723789;
   DATA[1936,31] := 1.281542;
   DATA[1936,32] := 0.7352687;
   DATA[1936,33] := 0.3083624;
   DATA[1936,34] := 2.0;
   DATA[1936,35] := 250.1762;
   DATA[1936,36] := 1.730048;
   DATA[1936,37] := 189.1022;
   DATA[1936,38] := 0.000128152;
   DATA[1936,39] := 1.0;
   DATA[1936,40] := 1.0;
   DATA[1937,0] := 2.497198;
   DATA[1937,1] := 860.813;
   DATA[1937,2] := 2.0;
   DATA[1937,3] := 2.0;
   DATA[1937,4] := 262.4648;
   DATA[1937,5] := 8.391951;
   DATA[1937,6] := 332.1969;
   DATA[1937,7] := 2.463333;
   DATA[1937,8] := 2.0;
   DATA[1937,9] := 2.0;
   DATA[1937,10] := 2.0;
   DATA[1937,11] := 19.73238;
   DATA[1937,12] := 2.208884;
   DATA[1937,13] := 795.5493;
   DATA[1937,14] := 1.0;
   DATA[1937,15] := 2.0;
   DATA[1937,16] := 1.0;
   DATA[1937,17] := 1.0;
   DATA[1937,18] := 1.0;
   DATA[1937,19] := 2.0;
   DATA[1937,20] := 148.808;
   DATA[1937,21] := 154.7552;
   DATA[1937,22] := 1.715183;
   DATA[1937,23] := 824.7501;
   DATA[1937,24] := 2.0;
   DATA[1937,25] := 2.0;
   DATA[1937,26] := 7.874135;
   DATA[1937,27] := 143.9375;
   DATA[1937,28] := 262.2404;
   DATA[1937,29] := 12.11228;
   DATA[1937,30] := 1.723789;
   DATA[1937,31] := 1.269117;
   DATA[1937,32] := 0.7352687;
   DATA[1937,33] := 0.3083624;
   DATA[1937,34] := 2.0;
   DATA[1937,35] := 250.1762;
   DATA[1937,36] := 1.730048;
   DATA[1937,37] := 189.1022;
   DATA[1937,38] := 0.000128152;
   DATA[1937,39] := 1.0;
   DATA[1937,40] := 1.0;
   DATA[1938,0] := 2.538513;
   DATA[1938,1] := 860.499;
   DATA[1938,2] := 2.0;
   DATA[1938,3] := 2.0;
   DATA[1938,4] := 262.4648;
   DATA[1938,5] := 8.391951;
   DATA[1938,6] := 332.1969;
   DATA[1938,7] := 2.463333;
   DATA[1938,8] := 2.0;
   DATA[1938,9] := 2.0;
   DATA[1938,10] := 2.0;
   DATA[1938,11] := 19.66195;
   DATA[1938,12] := 2.208884;
   DATA[1938,13] := 795.389;
   DATA[1938,14] := 1.0;
   DATA[1938,15] := 2.0;
   DATA[1938,16] := 1.0;
   DATA[1938,17] := 1.0;
   DATA[1938,18] := 1.0;
   DATA[1938,19] := 2.0;
   DATA[1938,20] := 148.808;
   DATA[1938,21] := 154.7552;
   DATA[1938,22] := 1.713389;
   DATA[1938,23] := 824.4424;
   DATA[1938,24] := 2.0;
   DATA[1938,25] := 2.0;
   DATA[1938,26] := 7.874135;
   DATA[1938,27] := 143.9375;
   DATA[1938,28] := 262.2404;
   DATA[1938,29] := 12.11228;
   DATA[1938,30] := 1.723789;
   DATA[1938,31] := 1.261432;
   DATA[1938,32] := 0.7352687;
   DATA[1938,33] := 0.3088108;
   DATA[1938,34] := 2.0;
   DATA[1938,35] := 250.1762;
   DATA[1938,36] := 1.730048;
   DATA[1938,37] := 189.1022;
   DATA[1938,38] := 0.000128152;
   DATA[1938,39] := 1.0;
   DATA[1938,40] := 1.0;
   DATA[1939,0] := 2.581751;
   DATA[1939,1] := 860.6559;
   DATA[1939,2] := 2.0;
   DATA[1939,3] := 2.0;
   DATA[1939,4] := 262.4648;
   DATA[1939,5] := 8.391951;
   DATA[1939,6] := 332.1969;
   DATA[1939,7] := 2.464614;
   DATA[1939,8] := 2.0;
   DATA[1939,9] := 2.0;
   DATA[1939,10] := 2.0;
   DATA[1939,11] := 19.66195;
   DATA[1939,12] := 2.208884;
   DATA[1939,13] := 795.7896;
   DATA[1939,14] := 1.0;
   DATA[1939,15] := 2.0;
   DATA[1939,16] := 1.0;
   DATA[1939,17] := 1.0;
   DATA[1939,18] := 1.0;
   DATA[1939,19] := 2.0;
   DATA[1939,20] := 148.808;
   DATA[1939,21] := 154.7552;
   DATA[1939,22] := 1.713389;
   DATA[1939,23] := 824.5963;
   DATA[1939,24] := 2.0;
   DATA[1939,25] := 2.0;
   DATA[1939,26] := 7.874135;
   DATA[1939,27] := 143.9375;
   DATA[1939,28] := 262.2404;
   DATA[1939,29] := 12.11228;
   DATA[1939,30] := 1.723789;
   DATA[1939,31] := 1.266171;
   DATA[1939,32] := 0.7352687;
   DATA[1939,33] := 0.3088108;
   DATA[1939,34] := 2.0;
   DATA[1939,35] := 250.1762;
   DATA[1939,36] := 1.730048;
   DATA[1939,37] := 189.022;
   DATA[1939,38] := 0.000128152;
   DATA[1939,39] := 1.0;
   DATA[1939,40] := 1.0;
   DATA[1940,0] := 2.618582;
   DATA[1940,1] := 860.5382;
   DATA[1940,2] := 2.0;
   DATA[1940,3] := 2.0;
   DATA[1940,4] := 262.4648;
   DATA[1940,5] := 8.391951;
   DATA[1940,6] := 332.1969;
   DATA[1940,7] := 2.464614;
   DATA[1940,8] := 2.0;
   DATA[1940,9] := 2.0;
   DATA[1940,10] := 2.0;
   DATA[1940,11] := 19.66195;
   DATA[1940,12] := 2.208884;
   DATA[1940,13] := 796.11;
   DATA[1940,14] := 1.0;
   DATA[1940,15] := 2.0;
   DATA[1940,16] := 1.0;
   DATA[1940,17] := 1.0;
   DATA[1940,18] := 1.0;
   DATA[1940,19] := 2.0;
   DATA[1940,20] := 148.808;
   DATA[1940,21] := 154.7552;
   DATA[1940,22] := 1.713389;
   DATA[1940,23] := 824.4809;
   DATA[1940,24] := 2.0;
   DATA[1940,25] := 2.0;
   DATA[1940,26] := 7.874135;
   DATA[1940,27] := 143.9375;
   DATA[1940,28] := 262.2404;
   DATA[1940,29] := 12.11228;
   DATA[1940,30] := 1.723789;
   DATA[1940,31] := 1.266428;
   DATA[1940,32] := 0.7352687;
   DATA[1940,33] := 0.3088108;
   DATA[1940,34] := 2.0;
   DATA[1940,35] := 250.1762;
   DATA[1940,36] := 1.730048;
   DATA[1940,37] := 189.022;
   DATA[1940,38] := 0.000128152;
   DATA[1940,39] := 1.0;
   DATA[1940,40] := 1.0;
   DATA[1941,0] := 2.649329;
   DATA[1941,1] := 860.2634;
   DATA[1941,2] := 2.0;
   DATA[1941,3] := 2.0;
   DATA[1941,4] := 262.4648;
   DATA[1941,5] := 8.391951;
   DATA[1941,6] := 332.1456;
   DATA[1941,7] := 2.464614;
   DATA[1941,8] := 2.0;
   DATA[1941,9] := 2.0;
   DATA[1941,10] := 2.0;
   DATA[1941,11] := 19.70357;
   DATA[1941,12] := 2.208884;
   DATA[1941,13] := 796.1901;
   DATA[1941,14] := 1.0;
   DATA[1941,15] := 2.0;
   DATA[1941,16] := 1.0;
   DATA[1941,17] := 1.0;
   DATA[1941,18] := 1.0;
   DATA[1941,19] := 2.0;
   DATA[1941,20] := 148.808;
   DATA[1941,21] := 154.7552;
   DATA[1941,22] := 1.712876;
   DATA[1941,23] := 824.6732;
   DATA[1941,24] := 2.0;
   DATA[1941,25] := 2.0;
   DATA[1941,26] := 7.874135;
   DATA[1941,27] := 143.9375;
   DATA[1941,28] := 262.0161;
   DATA[1941,29] := 12.11228;
   DATA[1941,30] := 1.723789;
   DATA[1941,31] := 1.268989;
   DATA[1941,32] := 0.7352687;
   DATA[1941,33] := 0.30785;
   DATA[1941,34] := 2.0;
   DATA[1941,35] := 250.1762;
   DATA[1941,36] := 1.730048;
   DATA[1941,37] := 189.022;
   DATA[1941,38] := 0.000128152;
   DATA[1941,39] := 1.0;
   DATA[1941,40] := 1.0;
   DATA[1942,0] := 2.655414;
   DATA[1942,1] := 860.5382;
   DATA[1942,2] := 2.0;
   DATA[1942,3] := 2.0;
   DATA[1942,4] := 262.4648;
   DATA[1942,5] := 8.391951;
   DATA[1942,6] := 332.0687;
   DATA[1942,7] := 2.464614;
   DATA[1942,8] := 2.0;
   DATA[1942,9] := 2.0;
   DATA[1942,10] := 2.0;
   DATA[1942,11] := 19.70357;
   DATA[1942,12] := 2.207091;
   DATA[1942,13] := 796.15;
   DATA[1942,14] := 1.0;
   DATA[1942,15] := 2.0;
   DATA[1942,16] := 1.0;
   DATA[1942,17] := 1.0;
   DATA[1942,18] := 1.0;
   DATA[1942,19] := 2.0;
   DATA[1942,20] := 148.808;
   DATA[1942,21] := 154.7552;
   DATA[1942,22] := 1.712876;
   DATA[1942,23] := 824.5963;
   DATA[1942,24] := 2.0;
   DATA[1942,25] := 2.0;
   DATA[1942,26] := 7.874135;
   DATA[1942,27] := 143.9375;
   DATA[1942,28] := 262.0161;
   DATA[1942,29] := 12.11228;
   DATA[1942,30] := 1.723789;
   DATA[1942,31] := 1.271679;
   DATA[1942,32] := 0.7352687;
   DATA[1942,33] := 0.30785;
   DATA[1942,34] := 2.0;
   DATA[1942,35] := 250.1762;
   DATA[1942,36] := 1.730048;
   DATA[1942,37] := 188.974;
   DATA[1942,38] := 0.000128152;
   DATA[1942,39] := 1.0;
   DATA[1942,40] := 1.0;
   DATA[1943,0] := 2.658617;
   DATA[1943,1] := 860.4205;
   DATA[1943,2] := 2.0;
   DATA[1943,3] := 2.0;
   DATA[1943,4] := 262.4648;
   DATA[1943,5] := 8.391951;
   DATA[1943,6] := 332.0687;
   DATA[1943,7] := 2.465767;
   DATA[1943,8] := 2.0;
   DATA[1943,9] := 2.0;
   DATA[1943,10] := 2.0;
   DATA[1943,11] := 19.71957;
   DATA[1943,12] := 2.207091;
   DATA[1943,13] := 796.7909;
   DATA[1943,14] := 1.0;
   DATA[1943,15] := 2.0;
   DATA[1943,16] := 1.0;
   DATA[1943,17] := 1.0;
   DATA[1943,18] := 1.0;
   DATA[1943,19] := 2.0;
   DATA[1943,20] := 148.808;
   DATA[1943,21] := 154.7552;
   DATA[1943,22] := 1.712876;
   DATA[1943,23] := 824.5963;
   DATA[1943,24] := 2.0;
   DATA[1943,25] := 2.0;
   DATA[1943,26] := 7.874135;
   DATA[1943,27] := 143.9375;
   DATA[1943,28] := 262.0161;
   DATA[1943,29] := 12.11228;
   DATA[1943,30] := 1.723789;
   DATA[1943,31] := 1.271679;
   DATA[1943,32] := 0.7352687;
   DATA[1943,33] := 0.30785;
   DATA[1943,34] := 2.0;
   DATA[1943,35] := 250.1762;
   DATA[1943,36] := 1.730048;
   DATA[1943,37] := 188.9259;
   DATA[1943,38] := 0.000128152;
   DATA[1943,39] := 1.0;
   DATA[1943,40] := 1.0;
   DATA[1944,0] := 2.651251;
   DATA[1944,1] := 860.342;
   DATA[1944,2] := 2.0;
   DATA[1944,3] := 2.0;
   DATA[1944,4] := 262.4648;
   DATA[1944,5] := 8.391951;
   DATA[1944,6] := 332.0687;
   DATA[1944,7] := 2.465767;
   DATA[1944,8] := 2.0;
   DATA[1944,9] := 2.0;
   DATA[1944,10] := 2.0;
   DATA[1944,11] := 19.73238;
   DATA[1944,12] := 2.207988;
   DATA[1944,13] := 796.7909;
   DATA[1944,14] := 1.0;
   DATA[1944,15] := 2.0;
   DATA[1944,16] := 1.0;
   DATA[1944,17] := 1.0;
   DATA[1944,18] := 1.0;
   DATA[1944,19] := 2.0;
   DATA[1944,20] := 148.808;
   DATA[1944,21] := 154.7552;
   DATA[1944,22] := 1.712876;
   DATA[1944,23] := 824.5963;
   DATA[1944,24] := 2.0;
   DATA[1944,25] := 2.0;
   DATA[1944,26] := 7.874135;
   DATA[1944,27] := 143.9375;
   DATA[1944,28] := 262.0161;
   DATA[1944,29] := 12.11228;
   DATA[1944,30] := 1.723789;
   DATA[1944,31] := 1.289868;
   DATA[1944,32] := 0.7352687;
   DATA[1944,33] := 0.3083624;
   DATA[1944,34] := 2.0;
   DATA[1944,35] := 250.1762;
   DATA[1944,36] := 1.730048;
   DATA[1944,37] := 188.8939;
   DATA[1944,38] := 0.000128152;
   DATA[1944,39] := 1.0;
   DATA[1944,40] := 1.0;
   DATA[1945,0] := 2.624988;
   DATA[1945,1] := 859.9102;
   DATA[1945,2] := 2.0;
   DATA[1945,3] := 2.0;
   DATA[1945,4] := 262.4648;
   DATA[1945,5] := 8.391951;
   DATA[1945,6] := 332.0687;
   DATA[1945,7] := 2.465767;
   DATA[1945,8] := 2.0;
   DATA[1945,9] := 2.0;
   DATA[1945,10] := 2.0;
   DATA[1945,11] := 19.73878;
   DATA[1945,12] := 2.207988;
   DATA[1945,13] := 797.3116;
   DATA[1945,14] := 1.0;
   DATA[1945,15] := 2.0;
   DATA[1945,16] := 1.0;
   DATA[1945,17] := 1.0;
   DATA[1945,18] := 1.0;
   DATA[1945,19] := 2.0;
   DATA[1945,20] := 148.808;
   DATA[1945,21] := 154.7552;
   DATA[1945,22] := 1.712876;
